Omron Sysmac Studio project Trabalho_Pratico1_vFinal_beta (Sysmac Studio 1.53.0.64009, StandardProject)

# Controller new_Controller_0: NX1P2-9B24DT1 version 1.42
Task PrimaryTask (priority 4, period or condition 4000): Tp1Automacao
Library OEN_Communication_V1_0_22 1.0.22 (contents left out)

VAR_GLOBAL RETAIN
    OutputsDigitais AT %D0 : ARRAY[0..150] OF BOOL;  (* Saidas Digitais; published *)
    DigitaInputs AT %D30 : ARRAY[0..150] OF BOOL;  (* Entradas Digitais; published *)
    AnalogInputs AT %D60 : ARRAY[0..25] OF WORD;  (* Entradas Analogicas; published *)
    AnalogOutput AT %D200 : ARRAY[0..25] OF WORD;  (* Saidas Analogicas; published *)
    Trama AT %D400 : ARRAY[0..5] OF OEN\Modbus\sModbusReq := [(Enable := True, NodeAdr := 1, FunctionCode := Fn02_ReadDiscreteInputs, Read := (StartAddressRemote := 0, StartAddressLocal := 0, Count := 35), Write := (StartAddressRemote := 0, StartAddressLocal := 0, Count := 0)), (Enable := False, NodeAdr := 1, FunctionCode := Fn05_WriteSingleCoil, Read := (StartAddressRemote := 0, StartAddressLocal := 0, Count := 0), Write := (StartAddressRemote := 0, StartAddressLocal := 0, Count := 40)), (Enable := True, NodeAdr := 1, FunctionCode := Fn15_WriteMultipleCoils, Read := (StartAddressRemote := 0, StartAddressLocal := 0, Count := 0), Write := (StartAddressRemote := 0, StartAddressLocal := 0, Count := 40)), (Enable := False, NodeAdr := 1, FunctionCode := Fn03_ReadHoldingRegisters, Read := (StartAddressRemote := 0, StartAddressLocal := 0, Count := 20), Write := (StartAddressRemote := 0, StartAddressLocal := 0, Count := 0)), (Enable := True, NodeAdr := 1, FunctionCode := Fn16_WriteMultipleRegisters, Read := (StartAddressRemote := 0, StartAddressLocal := 0, Count := 0), Write := (StartAddressRemote := 0, StartAddressLocal := 0, Count := 11)), (Enable := True, NodeAdr := 1, FunctionCode := Fn04_ReadInputRegisters, Read := (StartAddressRemote := 0, StartAddressLocal := 0, Count := 5), Write := (StartAddressRemote := 0, StartAddressLocal := 0, Count := 0))];  (* Trama de Comunicacao; published *)
END_VAR
VAR_GLOBAL
    Emerg_But : BOOL;  (* Botao de Emergencia; at BuiltInIO://cpu/#0/Input_Bit_01 *)
    Led_Is_On : BOOL;  (* Led Verde de Producao em Curso; at BuiltInIO://cpu/#0/Output_Bit_00 *)
    Start_But : BOOL;  (* Botao de início de linha; at BuiltInIO://cpu/#0/Input_Bit_02 *)
    Led_Is_Stop : BOOL;  (* Led Vermelho de linha parada; at BuiltInIO://cpu/#0/Output_Bit_01 *)
    Stop_But : BOOL;  (* Botao Stop- pára linha depois da caixa/peça ser removida; at BuiltInIO://cpu/#0/Input_Bit_03 *)
    Led_Is_Emergency : BOOL;  (* Led Amarelo de Emergência Ativa; at BuiltInIO://cpu/#0/Output_Bit_02 *)
    But_papel : BOOL;  (* Emite caixas de papel; at BuiltInIO://cpu/#0/Input_Bit_04 *)
    But_pecas : BOOL;  (* Emite peças azuis; at BuiltInIO://cpu/#0/Input_Bit_05 *)
    Sensor_IR : BOOL;  (* Sensor Infra Vermelho; at BuiltInIO://cpu/#0/Input_Bit_00 *)
    But_Reset : BOOL;  (* Reset aos contadores; at BuiltInIO://cpu/#0/Input_Bit_06 *)
    hmi_led_is_on AT %W0.00 : BOOL;  (* Led verde produção em curso; published *)
    hmi_led_is_emerg AT %W0.01 : BOOL;  (* Led amarelo de emergência; published *)
    hmi_led_is_stop AT %W0.02 : BOOL;  (* Led vermelho de linha parada; published *)
    hmi_StartBut AT %W0.03 : BOOL;  (* Botão Start- inicia linha; published *)
    hmi_StopBut AT %W0.04 : BOOL;  (* Botão Stop - pára linha depois da caixa/peça ser removida; published *)
    hmi_EmergBut AT %W0.05 : BOOL;  (* Botão Emergência - pára linha de imediato; published *)
    hmi_led_caixas AT %W0.06 : BOOL;  (* Led indica emissão de caixas de papel; published *)
    hmi_led_peças AT %W0.07 : BOOL;  (* Led indica emisão de peças azuis; published *)
    hmi_sw_emissor AT %W0.08 : BOOL;  (* Switch que emite peças (SW=0) ou caixas (SW=1); published *)
    hmi_resetCounter AT %W0.09 : BOOL;  (* Botão que dá reset aos contadores; published *)
    hmi_sw_kuka AT %W0.10 : BOOL;  (* SW=0 KUKA transforma peças em Base/ SW=1 "..."peças Lid; published *)
END_VAR
VAR_GLOBAL RETAIN
    hmi_pesoCaixa AT %D710 : INT;  (* Mostra peso da caixa; published *)
    hmi_alturaCaixa AT %D711 : INT;  (* Mostra altura da caixa; published *)
    hmi_Counter_Lid AT %D712 : INT;  (* Mosrador de peças Lid; published *)
    hmi_Counter_Base AT %D713 : INT;  (* Mostrador de peças Base; published *)
    hmi_Counter_S AT %D714 : INT;  (* Mostrador caixas S; published *)
    hmi_Counter_M AT %D715 : INT;  (* Mostrador caixas M; published *)
    hmi_Counter_L AT %D716 : INT;  (* Mostrador caixas L; published *)
END_VAR

PROGRAM Tp1Automacao
VAR
    Contact_Auxiliar : BOOL;  (* Active ad Desactive MODBUS *)
    Communication_Factory_IO : OEN\Modbus\ModbusTCP_Client;
    Etapas : INT := 0;  (* Etapas do Projeto *)
    timer_S4 : TON;  (* Permite uma leitura estável do valor medido na balança *)
END_VAR
VAR CONSTANT
    pesoCaixa_Ref : INT := 4;  (* Referencia de peso *)
END_VAR
VAR
    timer_S5 : TON;
END_VAR
VAR CONSTANT
    RightPP_Caixa1 : WORD := 8;  (* Posição em Volt para descer a Pick and Place *)
END_VAR
VAR
    timer_S6 : TON;
END_VAR
VAR RETAIN
    pesoCaixa : WORD;  (* guarda o valor do peso registado na balança *)
    pesoGuarda AT %D700 : INT;  (* Valor lido na balança em int *)
END_VAR
VAR
    ZaxisSetpoint_RightPP : WORD := 0;  (* Valor de referencia para descer o eixo Z da PP da Direita *)
    ZaxisSetpoint_KukaPP : WORD := 0;  (* Valor de referencia para descer o eixo Z da PP da kuka *)
END_VAR
VAR RETAIN
    alturaCaixa : WORD;  (* leitura o valor do altura *)
    alturaGuarda AT %D702 : INT;  (* guarda o valor da altura *)
END_VAR
VAR CONSTANT
    alturaCaixaRefM : INT := 192;  (* valor de ref para a caixa tamanho M *)
    alturaCaixaRefS : INT := 128;  (* valor de referencia para uma caixa de tamanho S (palletizing box) *)
    alturaCaixaRefL : INT := 224;  (* valor de referencia para uma caixa de tamanho L *)
    pesoCaixa_RefSmall : INT := 224;  (* ELIMINAR ESTA VARIAVEL *)
END_VAR
VAR
    timer_S7 : TON;  (* Tempo de Etiquetagem da Pick&Place Direita *)
    esteiraVel : WORD;  (* velocidade da esteira *)
    sensorVisaoLer : WORD;  (* Leitura do sensor de visão *)
END_VAR
VAR RETAIN
    sensorVisaoGuarda AT %D703 : INT;  (* guarda o valor do sensor de visao *)
END_VAR
VAR CONSTANT
    sensorVisaoRefLid : INT := 2;  (* Valor de referencia para uma tampa *)
    sensorVisaoRefRaw : INT := 1;  (* Valor de referencia para raw material *)
    sensorVisaoRefBase : INT := 3;  (* Valor de referencia para base *)
END_VAR
VAR RETAIN
    SBoxCountAux AT %D704 : INT := 0;  (* Contador de Caixas S *)
END_VAR
VAR
    SBoxCount : WORD;  (* Contador de Caixas S Para Automato *)
END_VAR
VAR RETAIN
    MBoxCountAux AT %D705 : INT := 0;  (* Contador de caixas M *)
END_VAR
VAR
    MBoxCount : WORD;  (* Contador de Caixas M Para Automato *)
END_VAR
VAR RETAIN
    LBoxCountAux AT %D706 : INT := 0;  (* Contador de caixas L *)
END_VAR
VAR
    LBoxCount : WORD;  (* Contador de Caixas L Para Automato *)
    timer_S8 : TON;  (* Tempo de atividade do Remover de Caixas S *)
    timer_S9 : TON;  (* Tempo de atividade do Remover de Caixas M *)
    timer_S10 : TON;  (* Tempo de atividade do Remover de Caixas L *)
END_VAR
VAR RETAIN
    ultimaEtapa AT %D707 : INT;  (* Variavel para guardar a ultima etapa *)
END_VAR
VAR
    ZaxisSetpoint_LeftPP : WORD := 0;  (* Valor de referencia para descer o eixo Z da PP da esquerda *)
    XaxisSetpoint_KukaPP : WORD := 0;  (* Movimento em X da pick and place *)
    timer_S11 : TON;  (* Tempo de Etiquetagem da Pick&Place Esquerda *)
END_VAR
VAR RETAIN
    LidCountAux AT %D708 : INT := 0;  (* Contador de Tampas *)
END_VAR
VAR
    LidCount : WORD;  (* Contador de Tampas para o LCD *)
END_VAR
VAR RETAIN
    BaseCountAux AT %D709 : INT := 0;  (* Contador de peças da base *)
END_VAR
VAR
    BaseCount : WORD;  (* Contador de peças base para o LCD *)
    timer_S12 : TON;  (* Tempo de atividade do Remover de Peças Lid *)
    timer_S13 : TON;  (* Tempo de atividade do Remover de Peças Base *)
    kukaSelect : INT := 0;
    ZaxisPosition_KukaPP : WORD := 0;
    XaxisPosition_KukaPP : WORD := 0;  (* Posição atual da Pick and Place da KUKA no eixo do X *)
    guardaPosZKuka : INT := 0;  (* Guarda o valor da PP da Kuka no eixo do Z *)
    guardaPosXKuka : INT := 0;  (* Guarda o valor da PP da Kuka no eixo do X *)
    SeletorKUKAAux : BOOL;  (* Variável que guarda o estado do seletor da KUKA *)
    timer_S14 : TON;  (* Permite a atualização de todos os contadores de materiais *)
    SeletorMaterialAux : BOOL;  (* Variável que guarda o estado do seletor de materiais (caixas= True / peças= False) *)
END_VAR
VAR_EXTERNAL
    OutputsDigitais : ARRAY[0..150] OF BOOL;  (* Saidas Digitais; [0] Emite peças azuis; [1] Conveyor de Entrada; [2] Conveyor da balança; [3] Ativador do Sorter; [5] Conveyor Direita; [4] Sorter Move para a Direita; [6] Sorter Move  para a Esquerda; [7] Conveyor da Esquerda; [8] Ativa tapete curvo direita; [9] Ativa tapete de medição de altura; [10] Pneumático caixa S; [11] Pneumático caixa M; [12] Pneumático caixa L; [13] Tapete curvo lado esquerdo; [14] Tapete zona de visão; [15] Vira o sorter para o raw material; [17] Vira o sorter para lid; [19] Vira o sorter para base; [16] Ativa o sorter para raw material; [18] Ativa o sorter para lid; [20] Ativa o sorter para base; [21] Tapete para a zona de separação peças; [24] Remover Caixas L; [23] Remover as Caixas do tamanho M; [22] Remover as caixas de tamanho S; [25] Conveyor de Transporte para KUKA; [27] Remover peças do tipo Base; [28] Remover peças do tipo Lid; [29] Emite caixas de papel; [30] Ativaçáo do Robot da KUKA; [31] Paragem do Robot da KUKA; [32] Conveyor Curvo da saida do Robot Kuka; [35] State=1 Ativar a fabricação de Lids. State=0 Ativar a fabricação de bases.; [36] Remover bases Kuka; [34] Tapete da direita após a saída da Kuka; [38] Agarrar na peça Pick and Place Kuka; [37] Remover tampas Kuka; [33] Conveyor lado das tampas Kuka; [39] Conveyor de Saida KUKA para peças *)
    DigitaInputs : ARRAY[0..150] OF BOOL;  (* Entradas Digitais; [0] IR Entrada; [1] Entrada na balança; [11] IR para ativar o tapete do sorter; [27] Seletor para a Kuka produzir bases; [2] IR Balança Meio; [3] IR Tapete Direita; [4] Sensor no local de etiquetagem (Direita); [5] IR Tapete Esquerda; [6] Sensor no Local de Etiquetagem (Esquerda); [7] Ativa o tapete curvo do lado direito; [8] Ativa o tapete de medição de altura; [9] IR de ativação do tapete curvo lado esquerdo; [10] IR de ativação do tapete zona de visão; [15] IR do pneumático das caixas S; [16] IR do pneumático das caixas M; [17] IR do pneumático das caixas L; [18] Deteção de caixa na pick and place da direita; [12] IR_Caixa na rampa tamanho S; [14] IR_Caixa na rampa tamanho L; [13] IR_Caixa na rampa tamanho M; [19] Detecao do Item na PP da Esquerda; [20] IR de entrada do conveyor da  KUKA; [21] Sensor do contador das bases; [22] Sensor do Contador das Lids; [23] Safety Door; [24] Sensor Capacitivo para entrada de peça producao do robot KUKA; [25] Sensor Capacitivo para notificar fim de producao de peças; [26] IR ativar o tapete apos a KUKA; [28] Seletor para a Kuka produzir Lids; [29] IR de separação de peças após a Kuka; [30] Sensor de proximidade da Pick and place da KUKA; [31] IR para contar tampas na parte da KUKA; [32] IR para contar bases na parte da kuka; [34] Estado do FactoryIO (Running ou não); [33] Estado do FactoryIO (Running ou não) *)
    AnalogInputs : ARRAY[0..25] OF WORD;  (* Entradas Analogicas; [0] Ler Peso; [1] AxisZ_Pos; [2] Sensor de visão; [3] Leitura de posição atual da Pick and Place em Z; [4] Leitura de posição atual da Pick and Place em X *)
    AnalogOutput : ARRAY[0..25] OF WORD;  (* Saidas Analogicas; [0] Esteira caixas de papelão / regular velocidade; [1] Posição do eixo Z da Pick&amp;Place Direita; [2] LCD do Contador de Caixas Pequemas ; [3] LCD das Caixas de tamanho M; [4] LCD das caixas de Tamanho L; [5] Eixo Z da PP da Esquerda; [7] Remover de peças to tipo Tampa; [8] Remover de peças to tipo Base; [9] Setpoint da posição para a pick and place da kuka Z; [10] Movimento Pick and Place KUKA em X *)
    Trama : ARRAY[0..5] OF OEN\Modbus\sModbusReq;  (* Trama de Comunicacao *)
    Start_But : BOOL;  (* Botao de inicio do tapete *)
    Led_Is_On : BOOL;  (* Led Verde de indicaçao de atividade *)
    Led_Is_Stop : BOOL;  (* Linha em Paragem *)
    Stop_But : BOOL;  (* Botao de Paragem da Producao *)
    Emerg_But : BOOL;
    Led_Is_Emergency : BOOL;
    But_papel : BOOL;  (* Botão que ativa emissão de caixas de papel- NO *)
    But_pecas : BOOL;  (* Botão que ativa a emissão de peças azuis- NC *)
    Sensor_IR : BOOL;  (* Sensor fisico IR *)
    But_Reset : BOOL;
    hmi_led_is_stop : BOOL;
    hmi_led_is_on : BOOL;
    hmi_pesoCaixa : INT;
    hmi_Counter_Lid : INT;
    hmi_Counter_Base : INT;
    hmi_Counter_S : INT;
    hmi_Counter_M : INT;
    hmi_Counter_L : INT;
    hmi_sw_kuka : BOOL;
    hmi_led_caixas : BOOL;
    hmi_led_peças : BOOL;
    hmi_resetCounter : BOOL;
    hmi_StartBut : BOOL;
    hmi_StopBut : BOOL;
    hmi_sw_emissor : BOOL;
    hmi_EmergBut : BOOL;
    hmi_alturaCaixa : INT;
    hmi_led_is_emerg : BOOL;
END_VAR
VAR
    _e1 : R_TRIG;
    _p2 : BOOL;
    _p3 : BOOL;
    _p4 : BOOL;
    _p5 : BOOL;
    _e6 : R_TRIG;
    _e7 : R_TRIG;
    _e8 : R_TRIG;
    _p9 : BOOL;
    _e10 : R_TRIG;
    _e11 : R_TRIG;
    _p12 : BOOL;
    _p13 : BOOL;
END_VAR

(* Section Tp1_Comunicação: ladder, written here as Structured Text *)

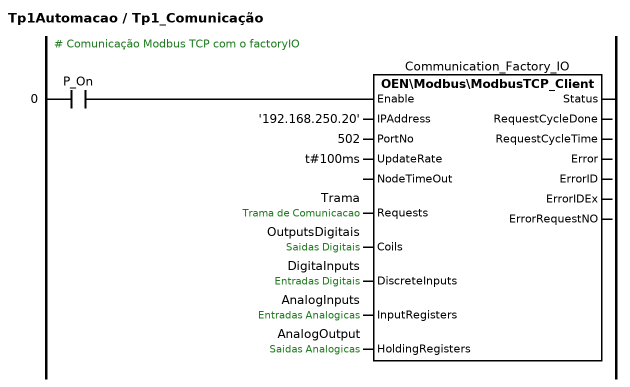
(* Rung 0: # Comunicação Modbus TCP com o factoryIO *)
Communication_Factory_IO(Enable := P_On, IPAddress := '192.168.250.20', PortNo := 502, UpdateRate := t#100ms, Requests := Trama, Coils := OutputsDigitais, DiscreteInputs := DigitaInputs, InputRegisters := AnalogInputs, HoldingRegisters := AnalogOutput);

(* Section Tp1_Botões: ladder, written here as Structured Text *)

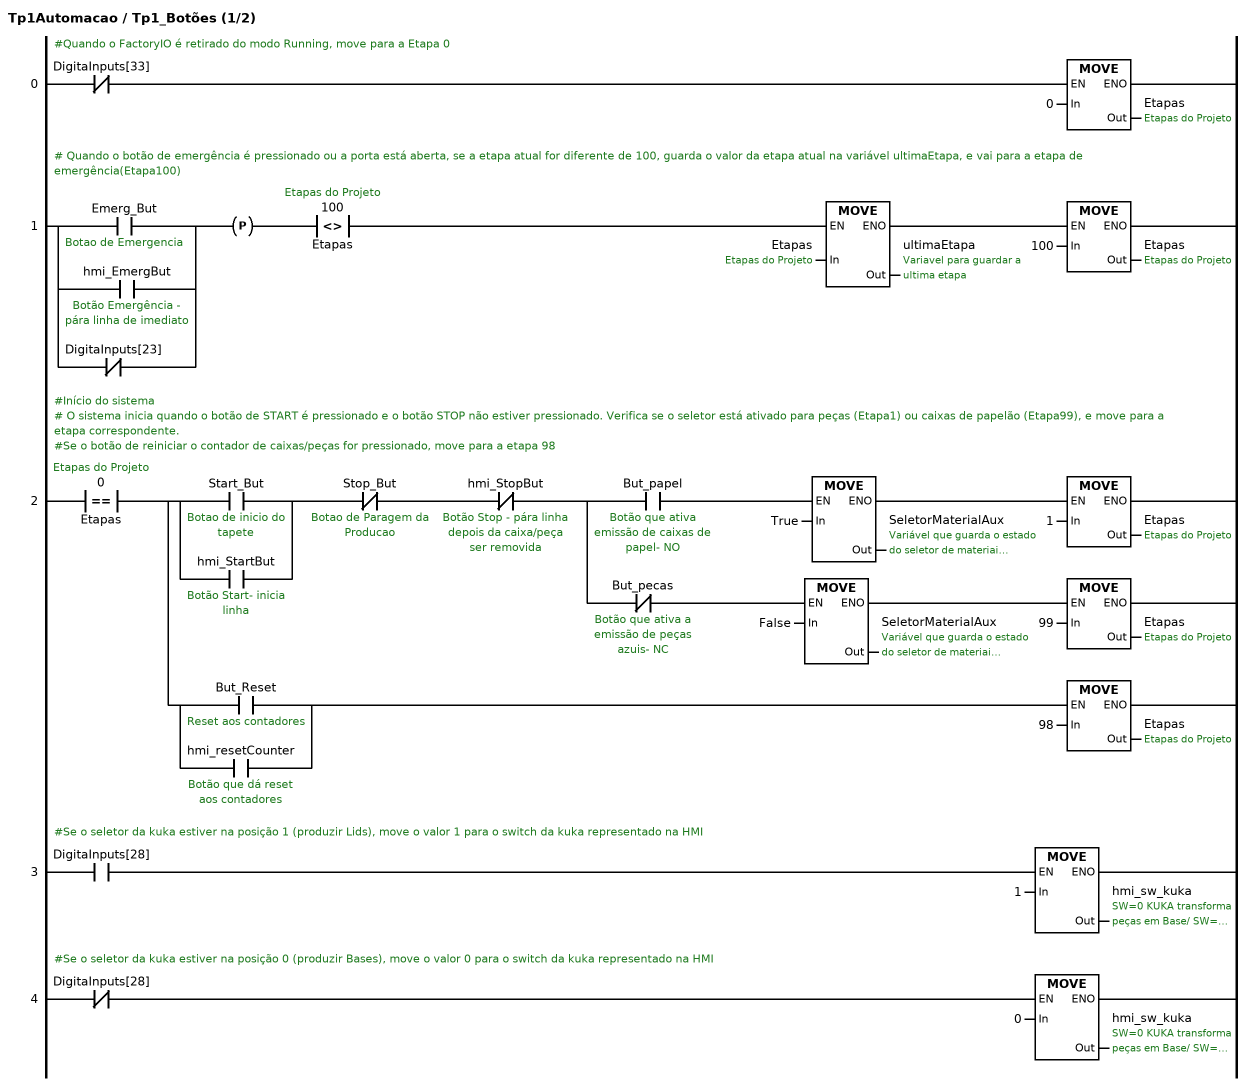
(* Rung 0: #Quando o FactoryIO é retirado do modo Running, move para a Etapa 0 *)
IF NOT DigitaInputs[33] THEN Etapas := 0; END_IF;
(* Rung 1: # Quando o botão de emergência é pressionado ou a porta está aberta, se a etapa atual for diferente de 100, guarda o valor da etapa atual na variável ultimaEtapa, e vai para a etapa de emergência(Etapa100) *)
_e1(CLK := Emerg_But OR hmi_EmergBut OR NOT DigitaInputs[23]);
IF _e1.Q AND (100 <> Etapas) THEN
    ultimaEtapa := Etapas;
    Etapas := 100;
END_IF;
(* Rung 2: #Início do sistema / # O sistema inicia quando o botão de START é pressionado e o botão STOP não estiver pressionado. Verifica se o seletor está ativado para peças (Etapa1) ou caixas de papelão (Etapa99), e move para a etapa correspondente. / #Se o botão de reiniciar o contador de caixas/peças for pressionado, move para a etapa 98 *)
_p2 := (0 = Etapas) AND (Start_But OR hmi_StartBut) AND NOT Stop_But AND NOT hmi_StopBut;
IF _p2 AND But_papel THEN SeletorMaterialAux := True; END_IF;
_p3 := 0 = Etapas;
IF _p2 AND But_papel THEN Etapas := 1; END_IF;
IF _p2 AND NOT But_pecas THEN
    SeletorMaterialAux := False;
    Etapas := 99;
END_IF;
IF _p3 AND (But_Reset OR hmi_resetCounter) THEN Etapas := 98; END_IF;
(* Rung 3: #Se o seletor da kuka estiver na posição 1 (produzir Lids), move o valor 1 para o switch da kuka representado na HMI *)
IF DigitaInputs[28] THEN hmi_sw_kuka := 1; END_IF;
(* Rung 4: #Se o seletor da kuka estiver na posição 0 (produzir Bases), move o valor 0 para o switch da kuka representado na HMI *)
IF NOT DigitaInputs[28] THEN hmi_sw_kuka := 0; END_IF;

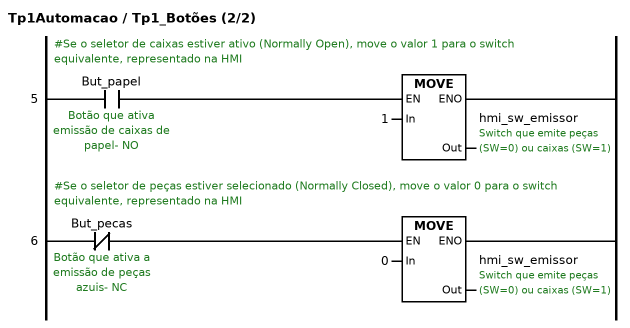
(* Rung 5: #Se o seletor de caixas estiver ativo (Normally Open), move o valor 1 para o switch equivalente, representado na HMI *)
IF But_papel THEN hmi_sw_emissor := 1; END_IF;
(* Rung 6: #Se o seletor de peças estiver selecionado (Normally Closed), move o valor 0 para o switch equivalente, representado na HMI *)
IF NOT But_pecas THEN hmi_sw_emissor := 0; END_IF;

(* Section Tp1_OutputsBotoes: ladder, written here as Structured Text *)

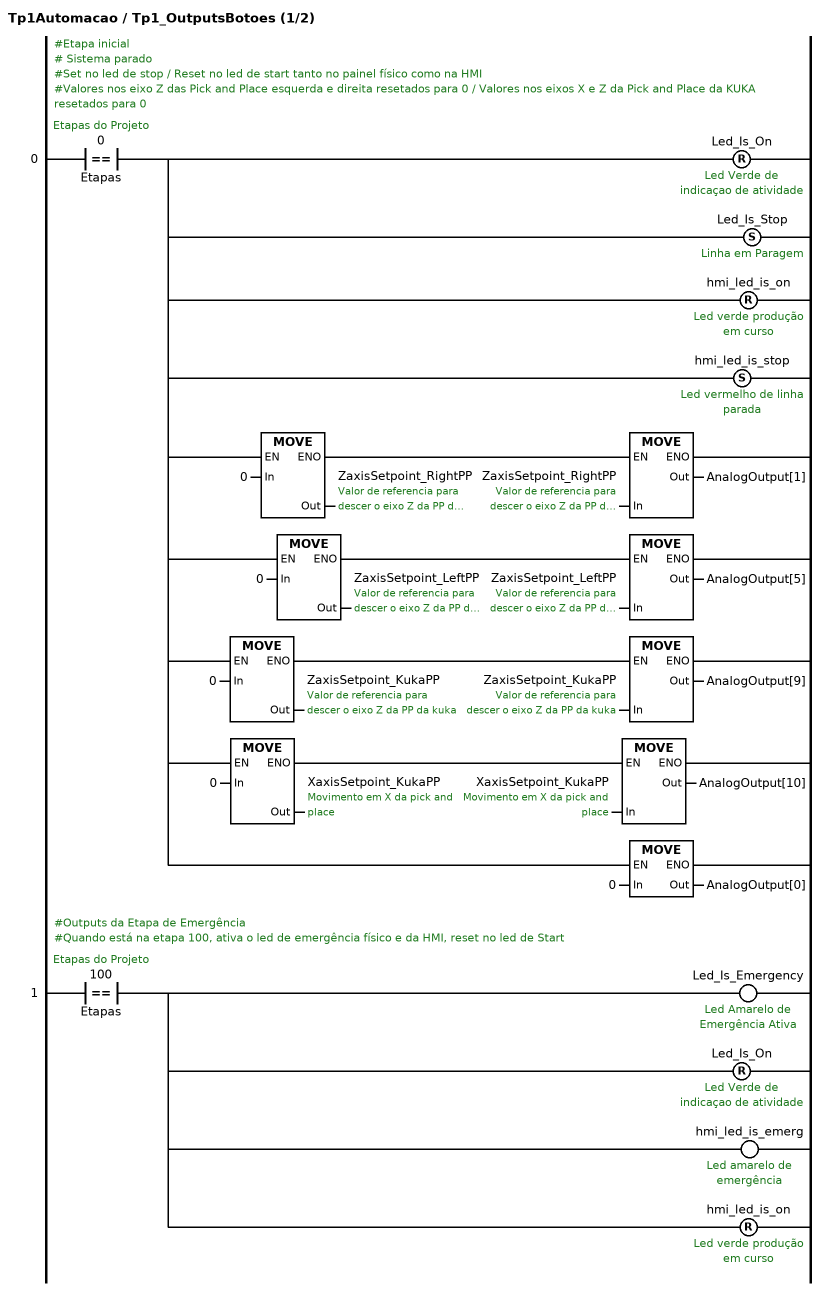
(* Rung 0: #Etapa inicial / # Sistema parado / #Set no led de stop / Reset no led de start tanto no painel físico como na HMI / #Valores nos eixo Z das Pick and Place esquerda e direita resetados para 0 / Valores nos eixos X e Z da Pick and Place da KUKA resetados para 0 *)
IF 0 = Etapas THEN
    Led_Is_On := FALSE;
    Led_Is_Stop := TRUE;
    hmi_led_is_on := FALSE;
    hmi_led_is_stop := TRUE;
    ZaxisSetpoint_RightPP := 0;
    AnalogOutput[1] := ZaxisSetpoint_RightPP;
    ZaxisSetpoint_LeftPP := 0;
    AnalogOutput[5] := ZaxisSetpoint_LeftPP;
    ZaxisSetpoint_KukaPP := 0;
    AnalogOutput[9] := ZaxisSetpoint_KukaPP;
    XaxisSetpoint_KukaPP := 0;
    AnalogOutput[10] := XaxisSetpoint_KukaPP;
    AnalogOutput[0] := 0;
END_IF;
(* Rung 1: #Outputs da Etapa de Emergência / #Quando está na etapa 100, ativa o led de emergência físico e da HMI, reset no led de Start *)
Led_Is_Emergency := 100 = Etapas;
IF 100 = Etapas THEN Led_Is_On := FALSE; END_IF;
hmi_led_is_emerg := 100 = Etapas;
IF 100 = Etapas THEN hmi_led_is_on := FALSE; END_IF;

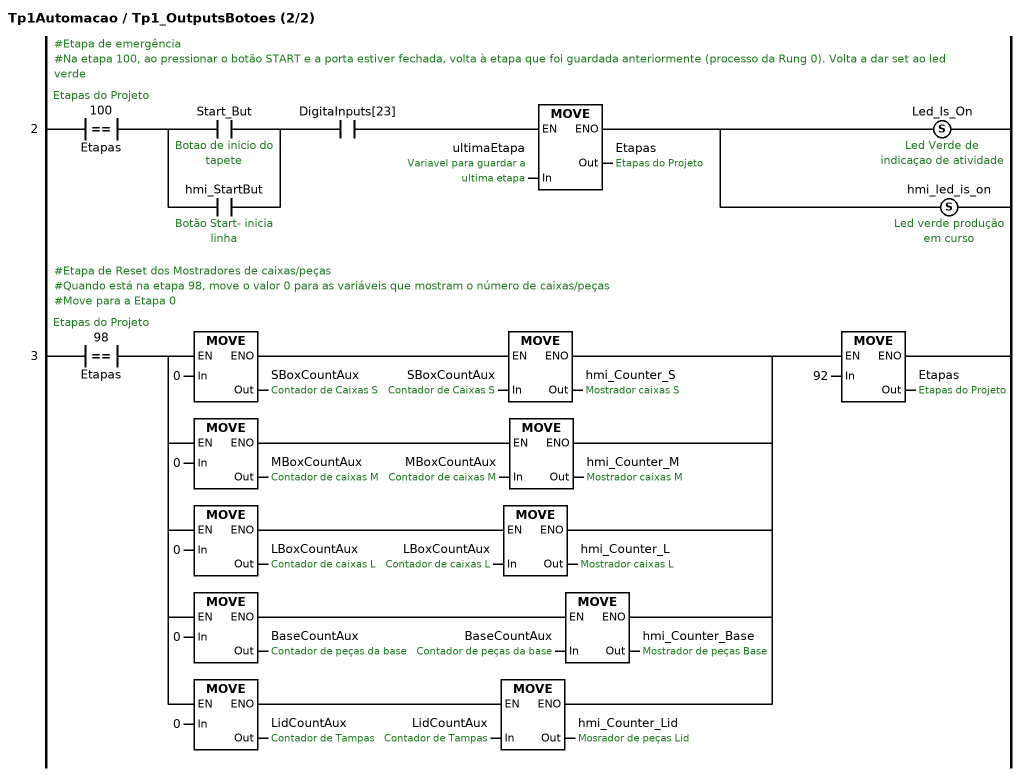
(* Rung 2: #Etapa de emergência / #Na etapa 100, ao pressionar o botão START e a porta estiver fechada, volta à etapa que foi guardada anteriormente (processo da Rung 0). Volta a dar set ao led verde *)
_p4 := (100 = Etapas) AND (Start_But OR hmi_StartBut) AND DigitaInputs[23];
IF _p4 THEN
    Etapas := ultimaEtapa;
    Led_Is_On := TRUE;
    hmi_led_is_on := TRUE;
END_IF;
(* Rung 3: #Etapa de Reset dos Mostradores de caixas/peças / #Quando está na etapa 98, move o valor 0 para as variáveis que mostram o número de caixas/peças / #Move para a Etapa 0 *)
IF 98 = Etapas THEN
    SBoxCountAux := 0;
    hmi_Counter_S := SBoxCountAux;
    MBoxCountAux := 0;
    hmi_Counter_M := MBoxCountAux;
    LBoxCountAux := 0;
    hmi_Counter_L := LBoxCountAux;
    BaseCountAux := 0;
    hmi_Counter_Base := BaseCountAux;
    LidCountAux := 0;
    hmi_Counter_Lid := LidCountAux;
    Etapas := 92;
END_IF;

(* Section Tp1_Etapas_ParteComum: ladder, written here as Structured Text *)

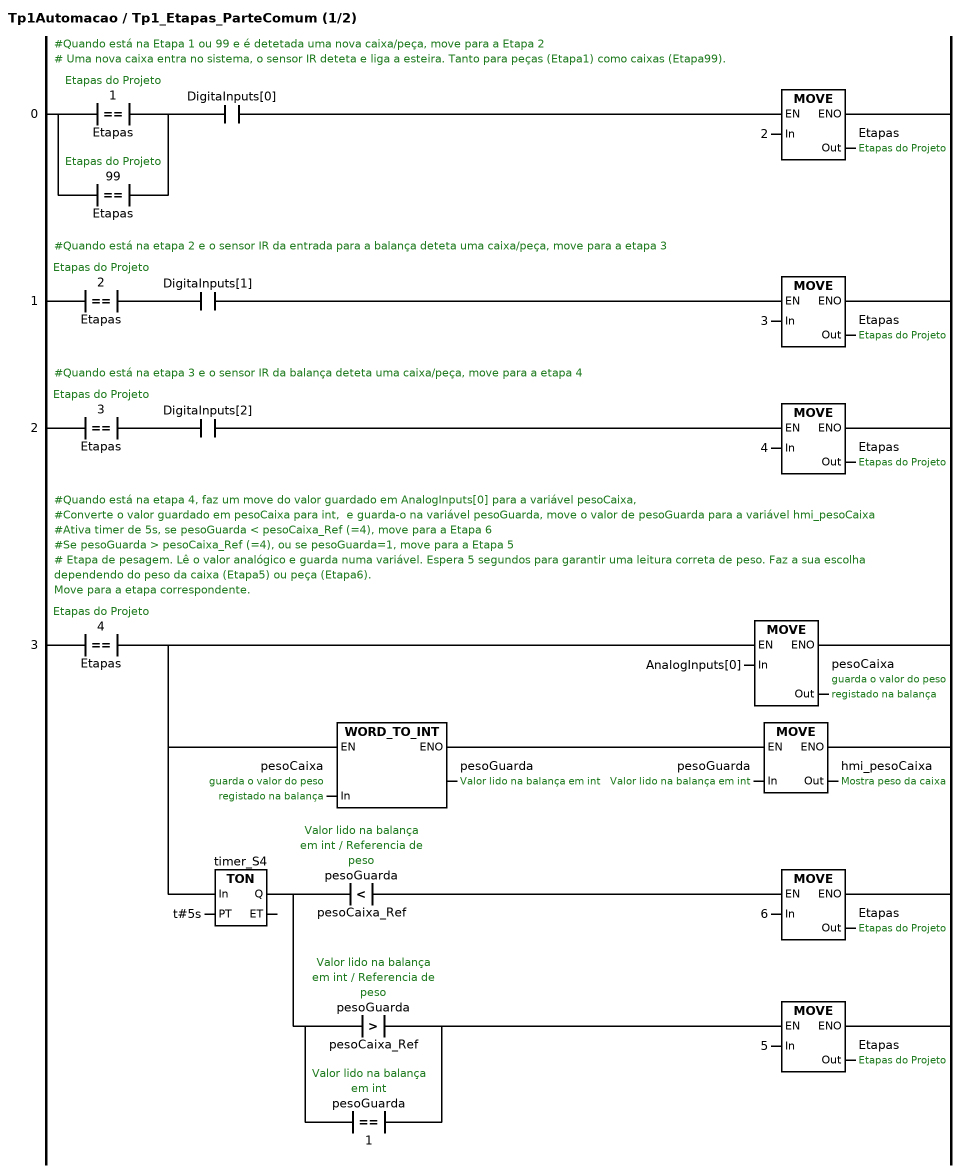
(* Rung 0: #Quando está na Etapa 1 ou 99 e é detetada uma nova caixa/peça, move para a Etapa 2 / # Uma nova caixa entra no sistema, o sensor IR deteta e liga a esteira. Tanto para peças (Etapa1) como caixas (Etapa99). *)
IF ((1 = Etapas) OR (99 = Etapas)) AND DigitaInputs[0] THEN Etapas := 2; END_IF;
(* Rung 1: #Quando está na etapa 2 e o sensor IR da entrada para a balança deteta uma caixa/peça, move para a etapa 3 *)
IF (2 = Etapas) AND DigitaInputs[1] THEN Etapas := 3; END_IF;
(* Rung 2: #Quando está na etapa 3 e o sensor IR da balança deteta uma caixa/peça, move para a etapa 4 *)
IF (3 = Etapas) AND DigitaInputs[2] THEN Etapas := 4; END_IF;
(* Rung 3: #Quando está na etapa 4, faz um move do valor guardado em AnalogInputs[0] para a variável pesoCaixa, / #Converte o valor guardado em pesoCaixa para int,  e guarda-o na variável pesoGuarda, move o valor de pesoGuarda para a variável hmi_pesoCaixa / #Ativa timer de 5s, se pesoGuarda < pesoCaixa_Ref (=4), move para a Etapa 6 / #Se pesoGuarda > pesoCaixa_Ref (=4), ou se pesoGuarda=1, move para a Etapa 5 / # Etapa de pesagem. Lê o valor analógico e guarda numa variável. Espera 5 segundos para garantir uma leitura correta de peso. Faz a sua escolha dependendo do peso da caixa (Etapa5) ou peça (Etapa6). / Move para a etapa correspondente. *)
IF 4 = Etapas THEN
    pesoCaixa := AnalogInputs[0];
    pesoGuarda := WORD_TO_INT(In := pesoCaixa);
    hmi_pesoCaixa := pesoGuarda;
END_IF;
timer_S4(In := 4 = Etapas, PT := t#5s);
IF timer_S4.Q AND (pesoGuarda < pesoCaixa_Ref) THEN Etapas := 6; END_IF;
IF timer_S4.Q AND ((pesoGuarda > pesoCaixa_Ref) OR (pesoGuarda = 1)) THEN Etapas := 5; END_IF;
(* notes on elements: #Permite a atualização de todos os contadores de materiais *)

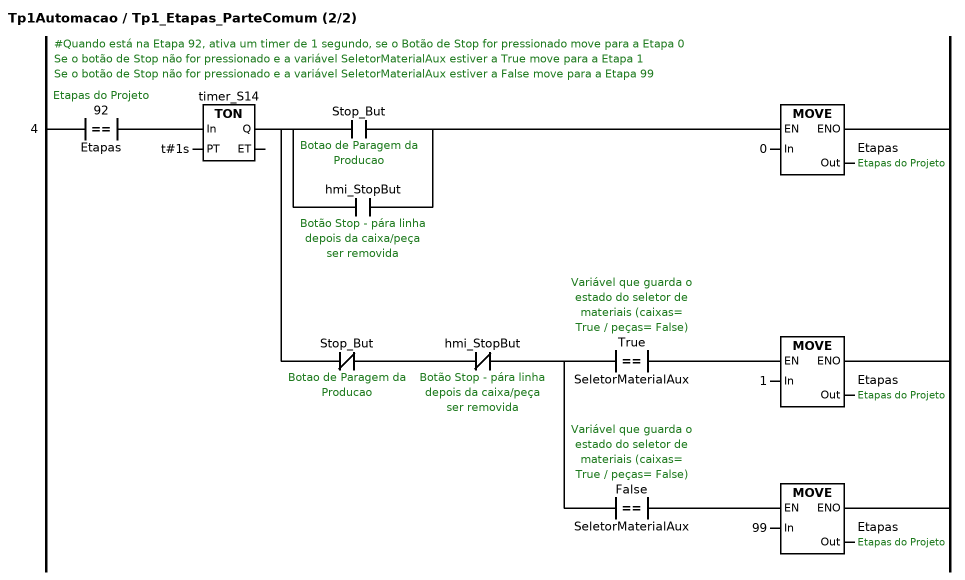
(* Rung 4: #Quando está na Etapa 92, ativa um timer de 1 segundo, se o Botão de Stop for pressionado move para a Etapa 0 / Se o botão de Stop não for pressionado e a variável SeletorMaterialAux estiver a True move para a Etapa 1 / Se o botão de Stop não for pressionado e a variável SeletorMaterialAux estiver a False move para a Etapa 99 *)
timer_S14(In := 92 = Etapas, PT := t#1s);
IF timer_S14.Q AND (Stop_But OR hmi_StopBut) THEN Etapas := 0; END_IF;
IF timer_S14.Q AND NOT Stop_But AND NOT hmi_StopBut AND (True = SeletorMaterialAux) THEN
    Etapas := 1;
END_IF;
IF timer_S14.Q AND NOT Stop_But AND NOT hmi_StopBut AND (False = SeletorMaterialAux) THEN
    Etapas := 99;
END_IF;
(* notes on elements: #Permite uma leitura estável do valor medido na balança *)

(* Section Tp1_Outputs_ParteComum: ladder, written here as Structured Text *)

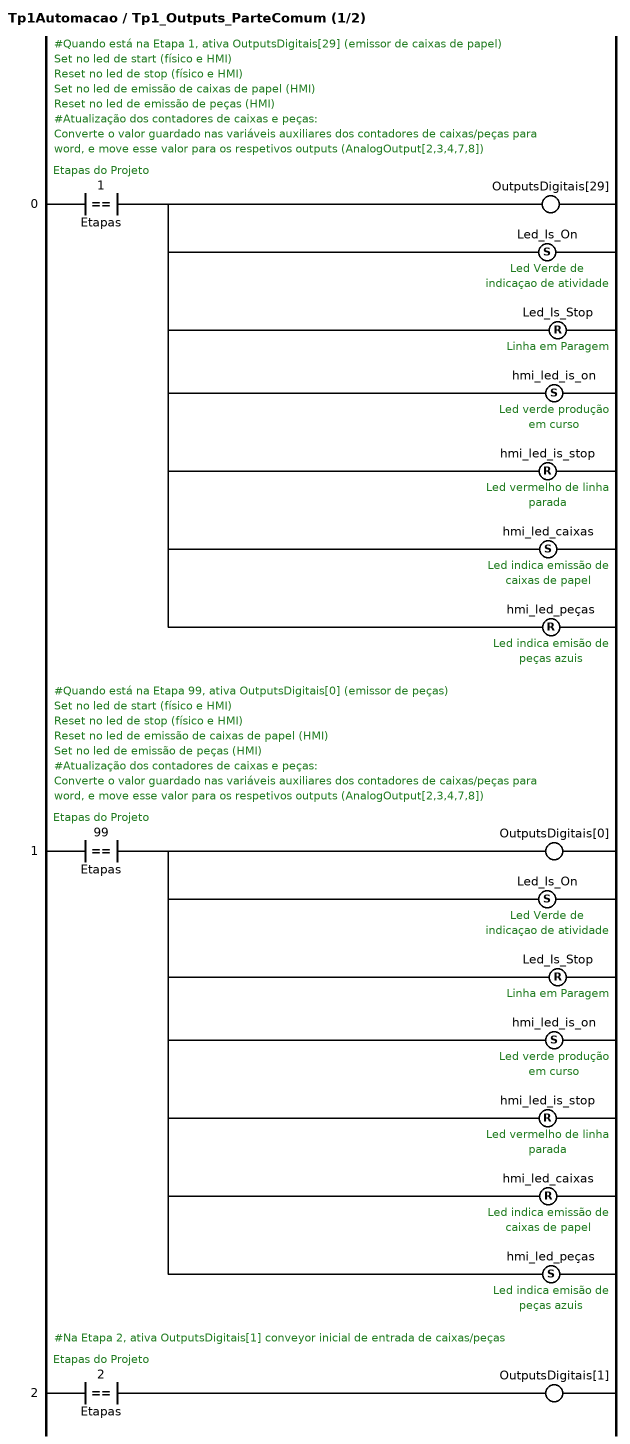
(* Rung 0: #Quando está na Etapa 1, ativa OutputsDigitais[29] (emissor de caixas de papel) / Set no led de start (físico e HMI) / Reset no led de stop (físico e HMI) / Set no led de emissão de caixas de papel (HMI) / Reset no led de emissão de peças (HMI) / #Atualização dos contadores de caixas e peças: / Converte o valor guardado nas variáveis auxiliares dos contadores de caixas/peças para word, e move esse valor para os respetivos outputs (AnalogOutput[2,3,4,7,8]) *)
OutputsDigitais[29] := 1 = Etapas;
IF 1 = Etapas THEN
    Led_Is_On := TRUE;
    Led_Is_Stop := FALSE;
    hmi_led_is_on := TRUE;
    hmi_led_is_stop := FALSE;
    hmi_led_caixas := TRUE;
    hmi_led_peças := FALSE;
END_IF;
(* Rung 1: #Quando está na Etapa 99, ativa OutputsDigitais[0] (emissor de peças) / Set no led de start (físico e HMI) / Reset no led de stop (físico e HMI) / Reset no led de emissão de caixas de papel (HMI) / Set no led de emissão de peças (HMI) / #Atualização dos contadores de caixas e peças: / Converte o valor guardado nas variáveis auxiliares dos contadores de caixas/peças para word, e move esse valor para os respetivos outputs (AnalogOutput[2,3,4,7,8]) *)
OutputsDigitais[0] := 99 = Etapas;
IF 99 = Etapas THEN
    Led_Is_On := TRUE;
    Led_Is_Stop := FALSE;
    hmi_led_is_on := TRUE;
    hmi_led_is_stop := FALSE;
    hmi_led_caixas := FALSE;
    hmi_led_peças := TRUE;
END_IF;
(* Rung 2: #Na Etapa 2, ativa OutputsDigitais[1] conveyor inicial de entrada de caixas/peças *)
OutputsDigitais[1] := 2 = Etapas;

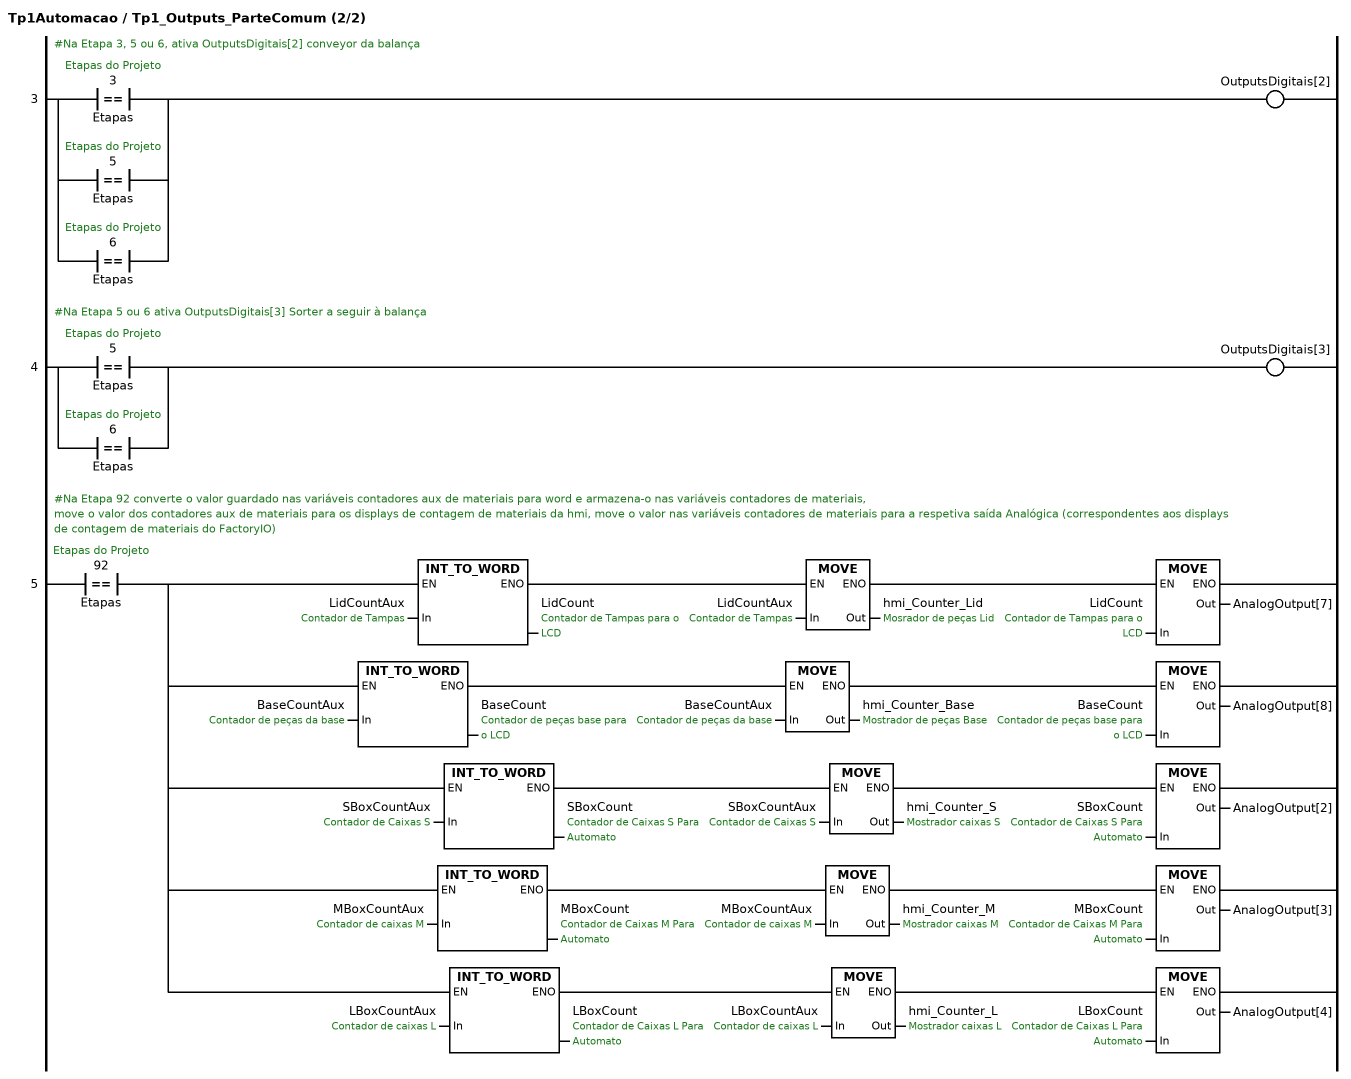
(* Rung 3: #Na Etapa 3, 5 ou 6, ativa OutputsDigitais[2] conveyor da balança *)
OutputsDigitais[2] := (3 = Etapas) OR (5 = Etapas) OR (6 = Etapas);
(* Rung 4: #Na Etapa 5 ou 6 ativa OutputsDigitais[3] Sorter a seguir à balança *)
OutputsDigitais[3] := (5 = Etapas) OR (6 = Etapas);
(* Rung 5: #Na Etapa 92 converte o valor guardado nas variáveis contadores aux de materiais para word e armazena-o nas variáveis contadores de materiais, / move o valor dos contadores aux de materiais para os displays de contagem de materiais da hmi, move o valor nas variáveis contadores de materiais para a respetiva saída Analógica (correspondentes aos displays / de contagem de materiais do FactoryIO) *)
IF 92 = Etapas THEN
    LidCount := INT_TO_WORD(In := LidCountAux);
    hmi_Counter_Lid := LidCountAux;
    AnalogOutput[7] := LidCount;
    BaseCount := INT_TO_WORD(In := BaseCountAux);
    hmi_Counter_Base := BaseCountAux;
    AnalogOutput[8] := BaseCount;
    SBoxCount := INT_TO_WORD(In := SBoxCountAux);
    hmi_Counter_S := SBoxCountAux;
    AnalogOutput[2] := SBoxCount;
    MBoxCount := INT_TO_WORD(In := MBoxCountAux);
    hmi_Counter_M := MBoxCountAux;
    AnalogOutput[3] := MBoxCount;
    LBoxCount := INT_TO_WORD(In := LBoxCountAux);
    hmi_Counter_L := LBoxCountAux;
    AnalogOutput[4] := LBoxCount;
END_IF;

(* Section Tp1_Etapas_ParteDireita: ladder, written here as Structured Text *)

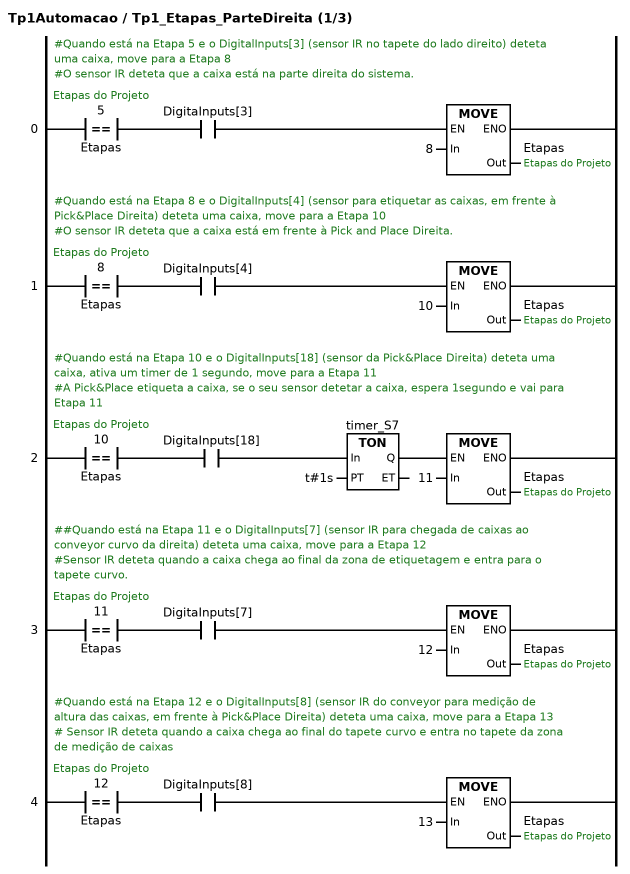
(* Rung 0: #Quando está na Etapa 5 e o DigitalInputs[3] (sensor IR no tapete do lado direito) deteta uma caixa, move para a Etapa 8 / #O sensor IR deteta que a caixa está na parte direita do sistema. *)
IF (5 = Etapas) AND DigitaInputs[3] THEN Etapas := 8; END_IF;
(* Rung 1: #Quando está na Etapa 8 e o DigitalInputs[4] (sensor para etiquetar as caixas, em frente à Pick&Place Direita) deteta uma caixa, move para a Etapa 10 / #O sensor IR deteta que a caixa está em frente à Pick and Place Direita. *)
IF (8 = Etapas) AND DigitaInputs[4] THEN Etapas := 10; END_IF;
(* Rung 2: #Quando está na Etapa 10 e o DigitalInputs[18] (sensor da Pick&Place Direita) deteta uma caixa, ativa um timer de 1 segundo, move para a Etapa 11 / #A Pick&Place etiqueta a caixa, se o seu sensor detetar a caixa, espera 1segundo e vai para Etapa 11 *)
timer_S7(In := (10 = Etapas) AND DigitaInputs[18], PT := t#1s);
IF timer_S7.Q THEN Etapas := 11; END_IF;
(* notes on elements: Tempo de Etiquetagem da Pick&Place Direita *)
(* Rung 3: ##Quando está na Etapa 11 e o DigitalInputs[7] (sensor IR para chegada de caixas ao conveyor curvo da direita) deteta uma caixa, move para a Etapa 12 / #Sensor IR deteta quando a caixa chega ao final da zona de etiquetagem e entra para o tapete curvo. *)
IF (11 = Etapas) AND DigitaInputs[7] THEN Etapas := 12; END_IF;
(* Rung 4: #Quando está na Etapa 12 e o DigitalInputs[8] (sensor IR do conveyor para medição de altura das caixas, em frente à Pick&Place Direita) deteta uma caixa, move para a Etapa 13 / # Sensor IR deteta quando a caixa chega ao final do tapete curvo e entra no tapete da zona de medição de caixas *)
IF (12 = Etapas) AND DigitaInputs[8] THEN Etapas := 13; END_IF;

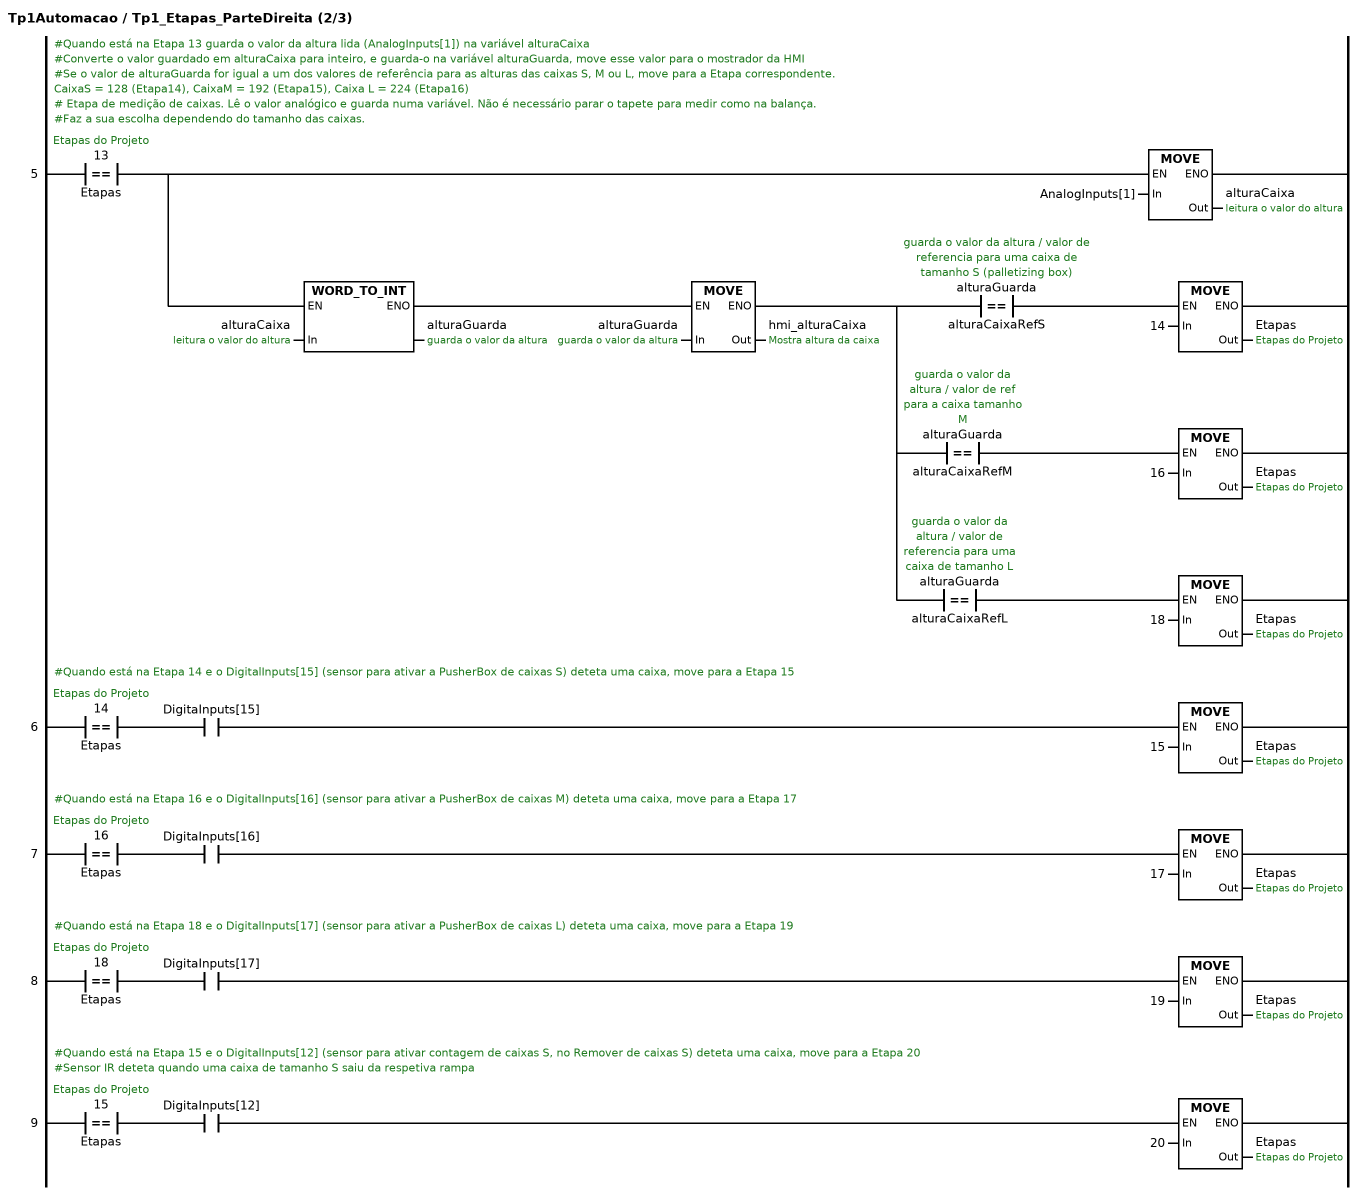
(* Rung 5: #Quando está na Etapa 13 guarda o valor da altura lida (AnalogInputs[1]) na variável alturaCaixa / #Converte o valor guardado em alturaCaixa para inteiro, e guarda-o na variável alturaGuarda, move esse valor para o mostrador da HMI / #Se o valor de alturaGuarda for igual a um dos valores de referência para as alturas das caixas S, M ou L, move para a Etapa correspondente. / CaixaS = 128 (Etapa14), CaixaM = 192 (Etapa15), Caixa L = 224 (Etapa16) / # Etapa de medição de caixas. Lê o valor analógico e guarda numa variável. Não é necessário parar o tapete para medir como na balança. / #Faz a sua escolha dependendo do tamanho das caixas. *)
IF 13 = Etapas THEN
    alturaCaixa := AnalogInputs[1];
    alturaGuarda := WORD_TO_INT(In := alturaCaixa);
    hmi_alturaCaixa := alturaGuarda;
END_IF;
_p5 := 13 = Etapas;
IF (13 = Etapas) AND (alturaGuarda = alturaCaixaRefS) THEN Etapas := 14; END_IF;
IF _p5 AND (alturaGuarda = alturaCaixaRefM) THEN Etapas := 16; END_IF;
IF _p5 AND (alturaGuarda = alturaCaixaRefL) THEN Etapas := 18; END_IF;
(* Rung 6: #Quando está na Etapa 14 e o DigitalInputs[15] (sensor para ativar a PusherBox de caixas S) deteta uma caixa, move para a Etapa 15 *)
IF (14 = Etapas) AND DigitaInputs[15] THEN Etapas := 15; END_IF;
(* Rung 7: #Quando está na Etapa 16 e o DigitalInputs[16] (sensor para ativar a PusherBox de caixas M) deteta uma caixa, move para a Etapa 17 *)
IF (16 = Etapas) AND DigitaInputs[16] THEN Etapas := 17; END_IF;
(* Rung 8: #Quando está na Etapa 18 e o DigitalInputs[17] (sensor para ativar a PusherBox de caixas L) deteta uma caixa, move para a Etapa 19 *)
IF (18 = Etapas) AND DigitaInputs[17] THEN Etapas := 19; END_IF;
(* Rung 9: #Quando está na Etapa 15 e o DigitalInputs[12] (sensor para ativar contagem de caixas S, no Remover de caixas S) deteta uma caixa, move para a Etapa 20 / #Sensor IR deteta quando uma caixa de tamanho S saiu da respetiva rampa *)
IF (15 = Etapas) AND DigitaInputs[12] THEN Etapas := 20; END_IF;

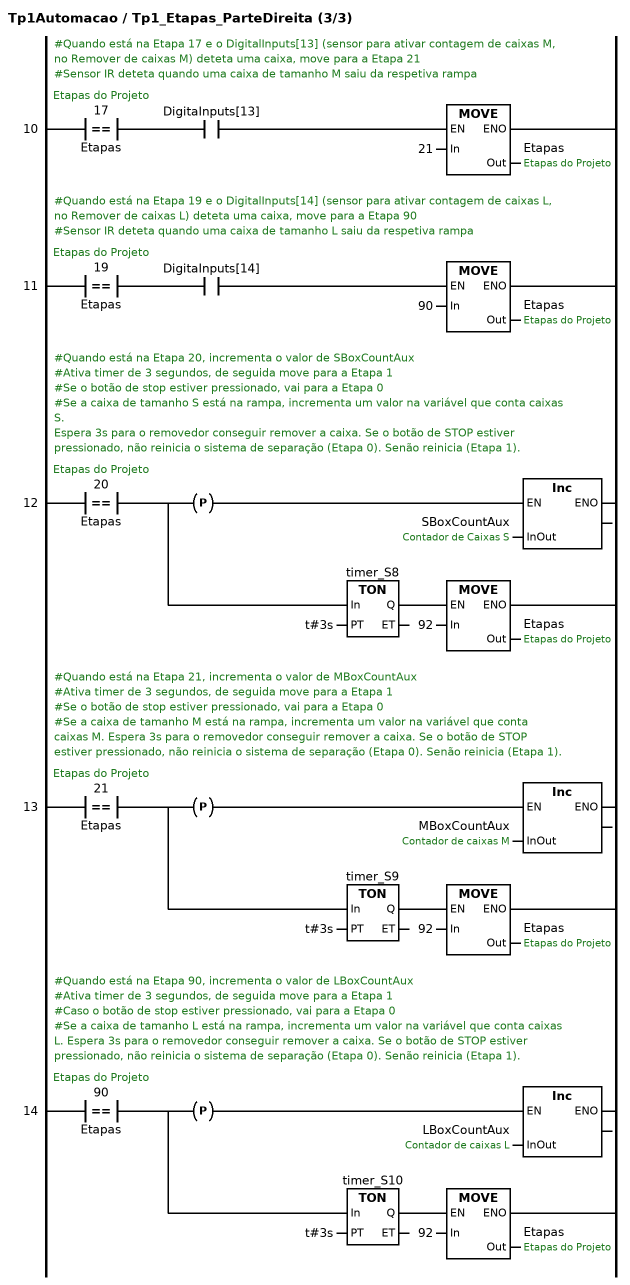
(* Rung 10: #Quando está na Etapa 17 e o DigitalInputs[13] (sensor para ativar contagem de caixas M, no Remover de caixas M) deteta uma caixa, move para a Etapa 21 / #Sensor IR deteta quando uma caixa de tamanho M saiu da respetiva rampa *)
IF (17 = Etapas) AND DigitaInputs[13] THEN Etapas := 21; END_IF;
(* Rung 11: #Quando está na Etapa 19 e o DigitalInputs[14] (sensor para ativar contagem de caixas L, no Remover de caixas L) deteta uma caixa, move para a Etapa 90 / #Sensor IR deteta quando uma caixa de tamanho L saiu da respetiva rampa *)
IF (19 = Etapas) AND DigitaInputs[14] THEN Etapas := 90; END_IF;
(* Rung 12: #Quando está na Etapa 20, incrementa o valor de SBoxCountAux / #Ativa timer de 3 segundos, de seguida move para a Etapa 1 / #Se o botão de stop estiver pressionado, vai para a Etapa 0 / #Se a caixa de tamanho S está na rampa, incrementa um valor na variável que conta caixas S. / Espera 3s para o removedor conseguir remover a caixa. Se o botão de STOP estiver pressionado, não reinicia o sistema de separação (Etapa 0). Senão reinicia (Etapa 1). *)
_e6(CLK := 20 = Etapas);
IF _e6.Q THEN Inc(InOut := SBoxCountAux); END_IF;
timer_S8(In := 20 = Etapas, PT := t#3s);
IF timer_S8.Q THEN Etapas := 92; END_IF;
(* notes on elements: Tempo de atividade do Remover de Caixas S *)
(* Rung 13: #Quando está na Etapa 21, incrementa o valor de MBoxCountAux / #Ativa timer de 3 segundos, de seguida move para a Etapa 1 / #Se o botão de stop estiver pressionado, vai para a Etapa 0 / #Se a caixa de tamanho M está na rampa, incrementa um valor na variável que conta caixas M. Espera 3s para o removedor conseguir remover a caixa. Se o botão de STOP estiver pressionado, não reinicia o sistema de separação (Etapa 0). Senão reinicia (Etapa 1). *)
_e7(CLK := 21 = Etapas);
IF _e7.Q THEN Inc(InOut := MBoxCountAux); END_IF;
timer_S9(In := 21 = Etapas, PT := t#3s);
IF timer_S9.Q THEN Etapas := 92; END_IF;
(* notes on elements: Tempo de atividade do Remover de Caixas M *)
(* Rung 14: #Quando está na Etapa 90, incrementa o valor de LBoxCountAux / #Ativa timer de 3 segundos, de seguida move para a Etapa 1 / #Caso o botão de stop estiver pressionado, vai para a Etapa 0 / #Se a caixa de tamanho L está na rampa, incrementa um valor na variável que conta caixas L. Espera 3s para o removedor conseguir remover a caixa. Se o botão de STOP estiver pressionado, não reinicia o sistema de separação (Etapa 0). Senão reinicia (Etapa 1). *)
_e8(CLK := 90 = Etapas);
IF _e8.Q THEN Inc(InOut := LBoxCountAux); END_IF;
timer_S10(In := 90 = Etapas, PT := t#3s);
IF timer_S10.Q THEN Etapas := 92; END_IF;
(* notes on elements: Tempo de atividade do Remover de Caixas L *)

(* Section Tp1_Outputs_ParteDireita: ladder, written here as Structured Text *)

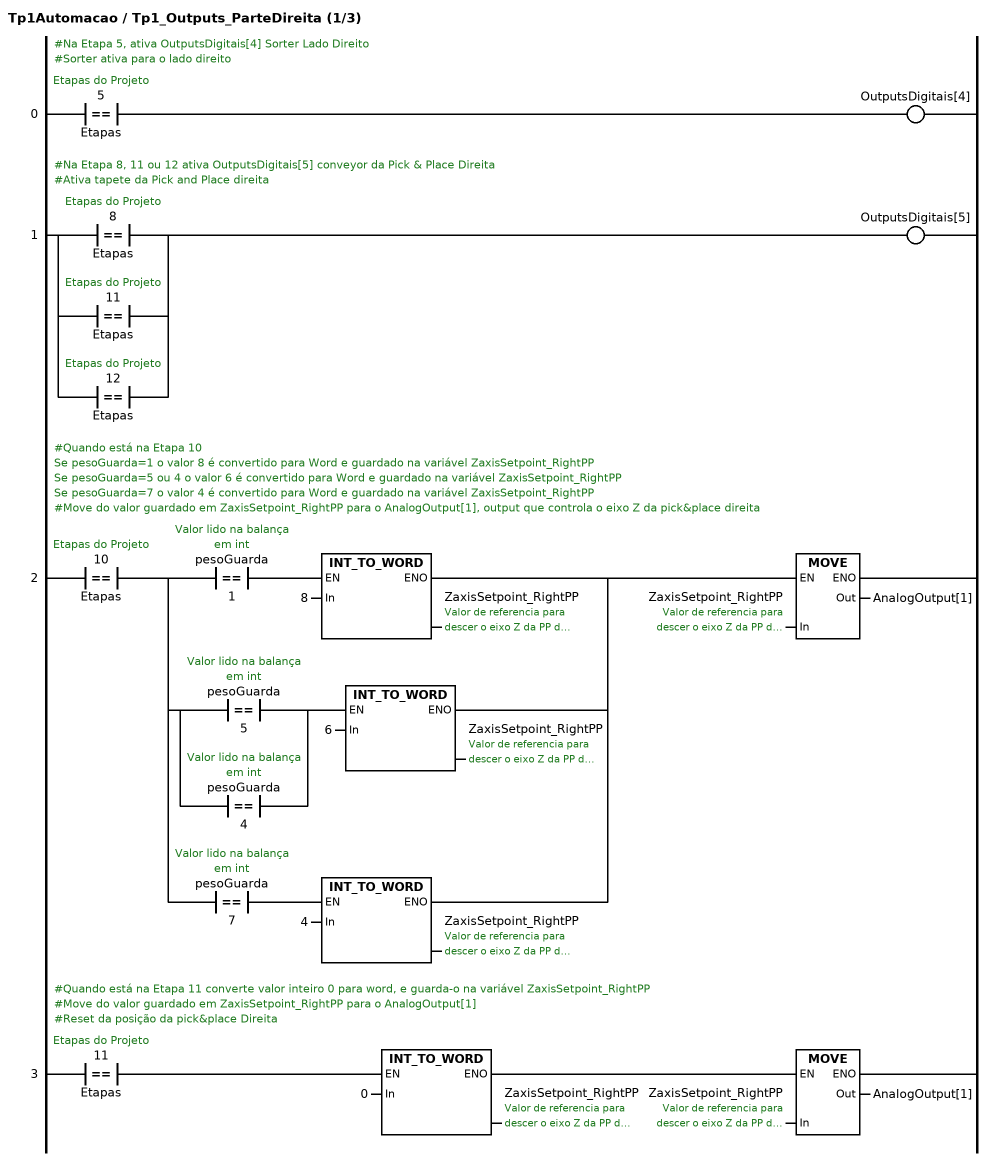
(* Rung 0: #Na Etapa 5, ativa OutputsDigitais[4] Sorter Lado Direito / #Sorter ativa para o lado direito *)
OutputsDigitais[4] := 5 = Etapas;
(* Rung 1: #Na Etapa 8, 11 ou 12 ativa OutputsDigitais[5] conveyor da Pick & Place Direita / #Ativa tapete da Pick and Place direita *)
OutputsDigitais[5] := (8 = Etapas) OR (11 = Etapas) OR (12 = Etapas);
(* Rung 2: #Quando está na Etapa 10 / Se pesoGuarda=1 o valor 8 é convertido para Word e guardado na variável ZaxisSetpoint_RightPP / Se pesoGuarda=5 ou 4 o valor 6 é convertido para Word e guardado na variável ZaxisSetpoint_RightPP / Se pesoGuarda=7 o valor 4 é convertido para Word e guardado na variável ZaxisSetpoint_RightPP / #Move do valor guardado em ZaxisSetpoint_RightPP para o AnalogOutput[1], output que controla o eixo Z da pick&place direita *)
IF (10 = Etapas) AND (pesoGuarda = 1) THEN ZaxisSetpoint_RightPP := INT_TO_WORD(In := 8); END_IF;
IF (10 = Etapas) AND ((pesoGuarda = 5) OR (pesoGuarda = 4)) THEN
    ZaxisSetpoint_RightPP := INT_TO_WORD(In := 6);
END_IF;
IF (10 = Etapas) AND (pesoGuarda = 7) THEN ZaxisSetpoint_RightPP := INT_TO_WORD(In := 4); END_IF;
IF (10 = Etapas) AND ((pesoGuarda = 1) OR (pesoGuarda = 5) OR (pesoGuarda = 4) OR (pesoGuarda = 7)) THEN
    AnalogOutput[1] := ZaxisSetpoint_RightPP;
END_IF;
(* Rung 3: #Quando está na Etapa 11 converte valor inteiro 0 para word, e guarda-o na variável ZaxisSetpoint_RightPP / #Move do valor guardado em ZaxisSetpoint_RightPP para o AnalogOutput[1] / #Reset da posição da pick&place Direita *)
IF 11 = Etapas THEN
    ZaxisSetpoint_RightPP := INT_TO_WORD(In := 0);
    AnalogOutput[1] := ZaxisSetpoint_RightPP;
END_IF;

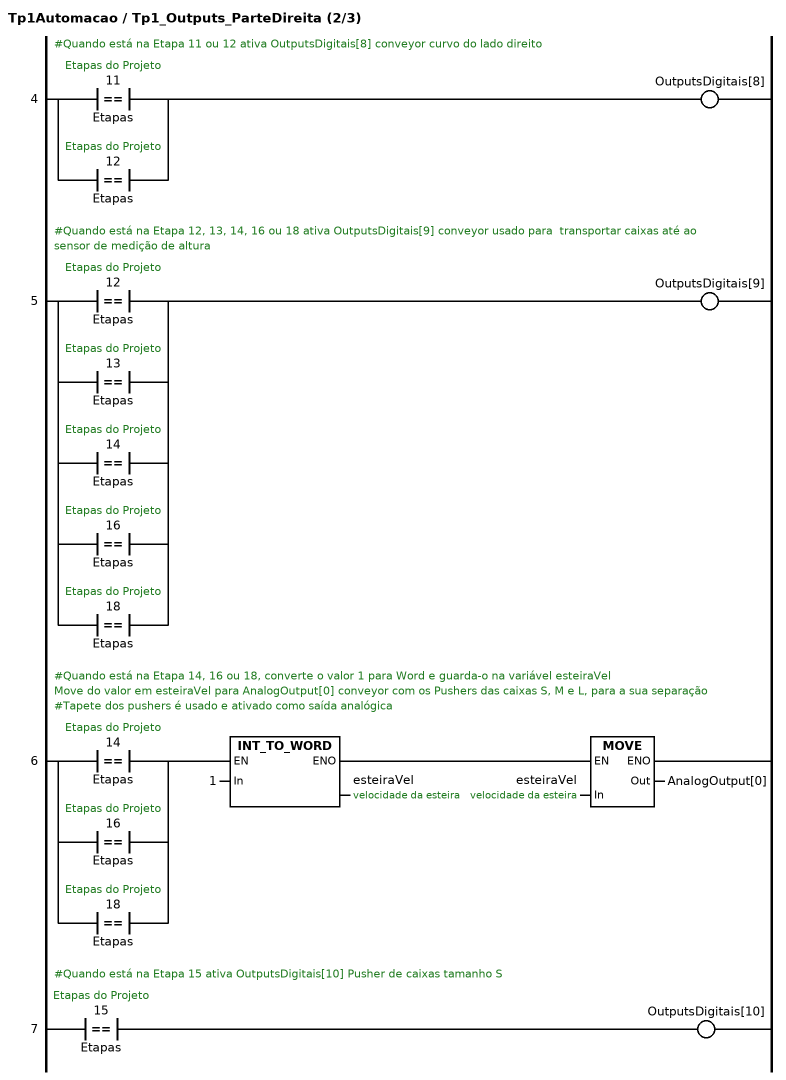
(* Rung 4: #Quando está na Etapa 11 ou 12 ativa OutputsDigitais[8] conveyor curvo do lado direito *)
OutputsDigitais[8] := (11 = Etapas) OR (12 = Etapas);
(* Rung 5: #Quando está na Etapa 12, 13, 14, 16 ou 18 ativa OutputsDigitais[9] conveyor usado para  transportar caixas até ao sensor de medição de altura *)
OutputsDigitais[9] := (12 = Etapas) OR (13 = Etapas) OR (14 = Etapas) OR (16 = Etapas) OR (18 = Etapas);
(* Rung 6: #Quando está na Etapa 14, 16 ou 18, converte o valor 1 para Word e guarda-o na variável esteiraVel / Move do valor em esteiraVel para AnalogOutput[0] conveyor com os Pushers das caixas S, M e L, para a sua separação / #Tapete dos pushers é usado e ativado como saída analógica *)
IF (14 = Etapas) OR (16 = Etapas) OR (18 = Etapas) THEN
    esteiraVel := INT_TO_WORD(In := 1);
    AnalogOutput[0] := esteiraVel;
END_IF;
(* Rung 7: #Quando está na Etapa 15 ativa OutputsDigitais[10] Pusher de caixas tamanho S *)
OutputsDigitais[10] := 15 = Etapas;

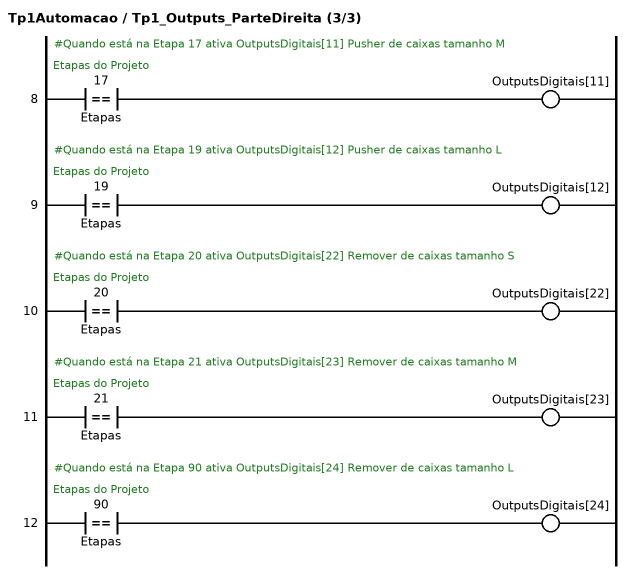
(* Rung 8: #Quando está na Etapa 17 ativa OutputsDigitais[11] Pusher de caixas tamanho M *)
OutputsDigitais[11] := 17 = Etapas;
(* Rung 9: #Quando está na Etapa 19 ativa OutputsDigitais[12] Pusher de caixas tamanho L *)
OutputsDigitais[12] := 19 = Etapas;
(* Rung 10: #Quando está na Etapa 20 ativa OutputsDigitais[22] Remover de caixas tamanho S *)
OutputsDigitais[22] := 20 = Etapas;
(* Rung 11: #Quando está na Etapa 21 ativa OutputsDigitais[23] Remover de caixas tamanho M *)
OutputsDigitais[23] := 21 = Etapas;
(* Rung 12: #Quando está na Etapa 90 ativa OutputsDigitais[24] Remover de caixas tamanho L *)
OutputsDigitais[24] := 90 = Etapas;

(* Section Tp1_Etapas_ParteEsquerda: ladder, written here as Structured Text *)

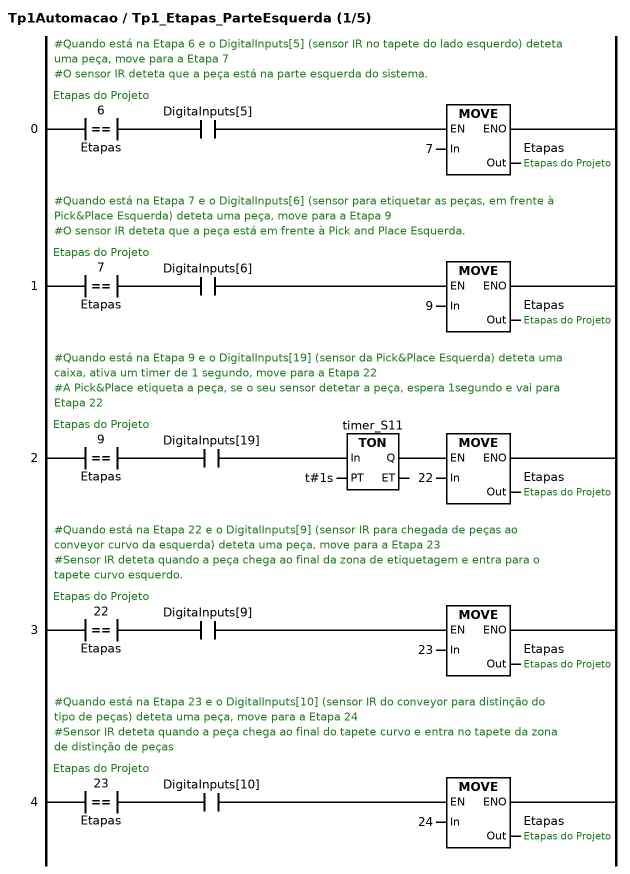
(* Rung 0: #Quando está na Etapa 6 e o DigitalInputs[5] (sensor IR no tapete do lado esquerdo) deteta uma peça, move para a Etapa 7 / #O sensor IR deteta que a peça está na parte esquerda do sistema. *)
IF (6 = Etapas) AND DigitaInputs[5] THEN Etapas := 7; END_IF;
(* Rung 1: #Quando está na Etapa 7 e o DigitalInputs[6] (sensor para etiquetar as peças, em frente à Pick&Place Esquerda) deteta uma peça, move para a Etapa 9 / #O sensor IR deteta que a peça está em frente à Pick and Place Esquerda. *)
IF (7 = Etapas) AND DigitaInputs[6] THEN Etapas := 9; END_IF;
(* Rung 2: #Quando está na Etapa 9 e o DigitalInputs[19] (sensor da Pick&Place Esquerda) deteta uma caixa, ativa um timer de 1 segundo, move para a Etapa 22 / #A Pick&Place etiqueta a peça, se o seu sensor detetar a peça, espera 1segundo e vai para Etapa 22 *)
timer_S11(In := (9 = Etapas) AND DigitaInputs[19], PT := t#1s);
IF timer_S11.Q THEN Etapas := 22; END_IF;
(* notes on elements: Tempo de Etiquetagem da Pick&Place Esquerda *)
(* Rung 3: #Quando está na Etapa 22 e o DigitalInputs[9] (sensor IR para chegada de peças ao conveyor curvo da esquerda) deteta uma peça, move para a Etapa 23 / #Sensor IR deteta quando a peça chega ao final da zona de etiquetagem e entra para o tapete curvo esquerdo. *)
IF (22 = Etapas) AND DigitaInputs[9] THEN Etapas := 23; END_IF;
(* Rung 4: #Quando está na Etapa 23 e o DigitalInputs[10] (sensor IR do conveyor para distinção do tipo de peças) deteta uma peça, move para a Etapa 24 / #Sensor IR deteta quando a peça chega ao final do tapete curvo e entra no tapete da zona de distinção de peças *)
IF (23 = Etapas) AND DigitaInputs[10] THEN Etapas := 24; END_IF;

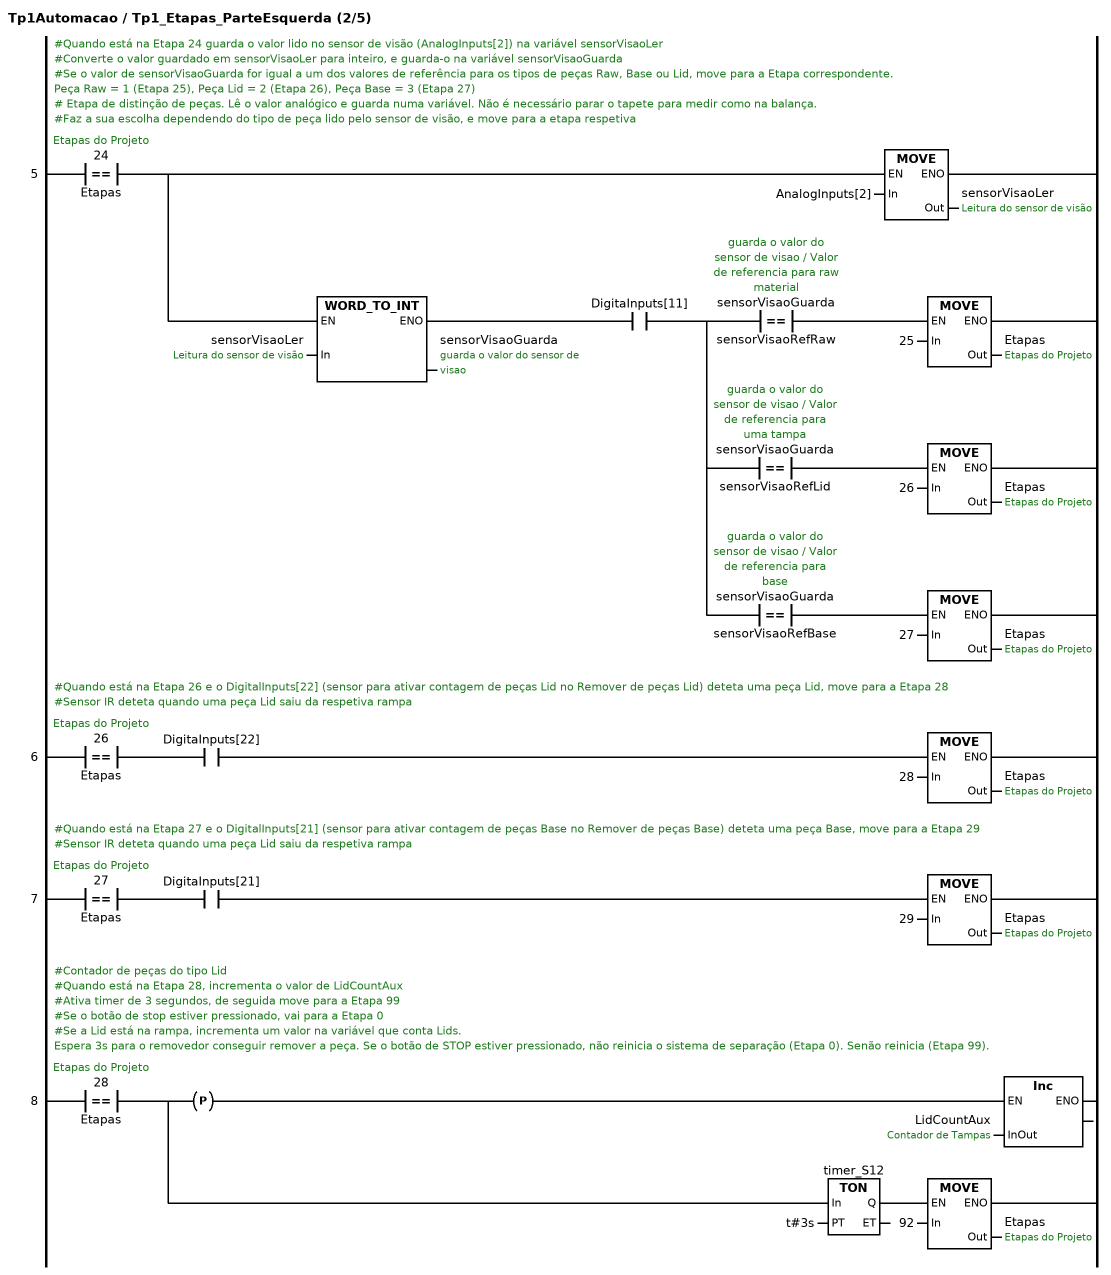
(* Rung 5: #Quando está na Etapa 24 guarda o valor lido no sensor de visão (AnalogInputs[2]) na variável sensorVisaoLer / #Converte o valor guardado em sensorVisaoLer para inteiro, e guarda-o na variável sensorVisaoGuarda / #Se o valor de sensorVisaoGuarda for igual a um dos valores de referência para os tipos de peças Raw, Base ou Lid, move para a Etapa correspondente. / Peça Raw = 1 (Etapa 25), Peça Lid = 2 (Etapa 26), Peça Base = 3 (Etapa 27) / # Etapa de distinção de peças. Lê o valor analógico e guarda numa variável. Não é necessário parar o tapete para medir como na balança. / #Faz a sua escolha dependendo do tipo de peça lido pelo sensor de visão, e move para a etapa respetiva *)
IF 24 = Etapas THEN
    sensorVisaoLer := AnalogInputs[2];
    sensorVisaoGuarda := WORD_TO_INT(In := sensorVisaoLer);
END_IF;
_p9 := (24 = Etapas) AND DigitaInputs[11];
IF (24 = Etapas) AND DigitaInputs[11] AND (sensorVisaoGuarda = sensorVisaoRefRaw) THEN
    Etapas := 25;
END_IF;
IF _p9 AND (sensorVisaoGuarda = sensorVisaoRefLid) THEN Etapas := 26; END_IF;
IF _p9 AND (sensorVisaoGuarda = sensorVisaoRefBase) THEN Etapas := 27; END_IF;
(* Rung 6: #Quando está na Etapa 26 e o DigitalInputs[22] (sensor para ativar contagem de peças Lid no Remover de peças Lid) deteta uma peça Lid, move para a Etapa 28 / #Sensor IR deteta quando uma peça Lid saiu da respetiva rampa *)
IF (26 = Etapas) AND DigitaInputs[22] THEN Etapas := 28; END_IF;
(* Rung 7: #Quando está na Etapa 27 e o DigitalInputs[21] (sensor para ativar contagem de peças Base no Remover de peças Base) deteta uma peça Base, move para a Etapa 29 / #Sensor IR deteta quando uma peça Lid saiu da respetiva rampa *)
IF (27 = Etapas) AND DigitaInputs[21] THEN Etapas := 29; END_IF;
(* Rung 8: #Contador de peças do tipo Lid / #Quando está na Etapa 28, incrementa o valor de LidCountAux / #Ativa timer de 3 segundos, de seguida move para a Etapa 99 / #Se o botão de stop estiver pressionado, vai para a Etapa 0 / #Se a Lid está na rampa, incrementa um valor na variável que conta Lids. / Espera 3s para o removedor conseguir remover a peça. Se o botão de STOP estiver pressionado, não reinicia o sistema de separação (Etapa 0). Senão reinicia (Etapa 99). *)
_e10(CLK := 28 = Etapas);
IF _e10.Q THEN Inc(InOut := LidCountAux); END_IF;
timer_S12(In := 28 = Etapas, PT := t#3s);
IF timer_S12.Q THEN Etapas := 92; END_IF;
(* notes on elements: Tempo de atividade do Remover de Peças Lid *)

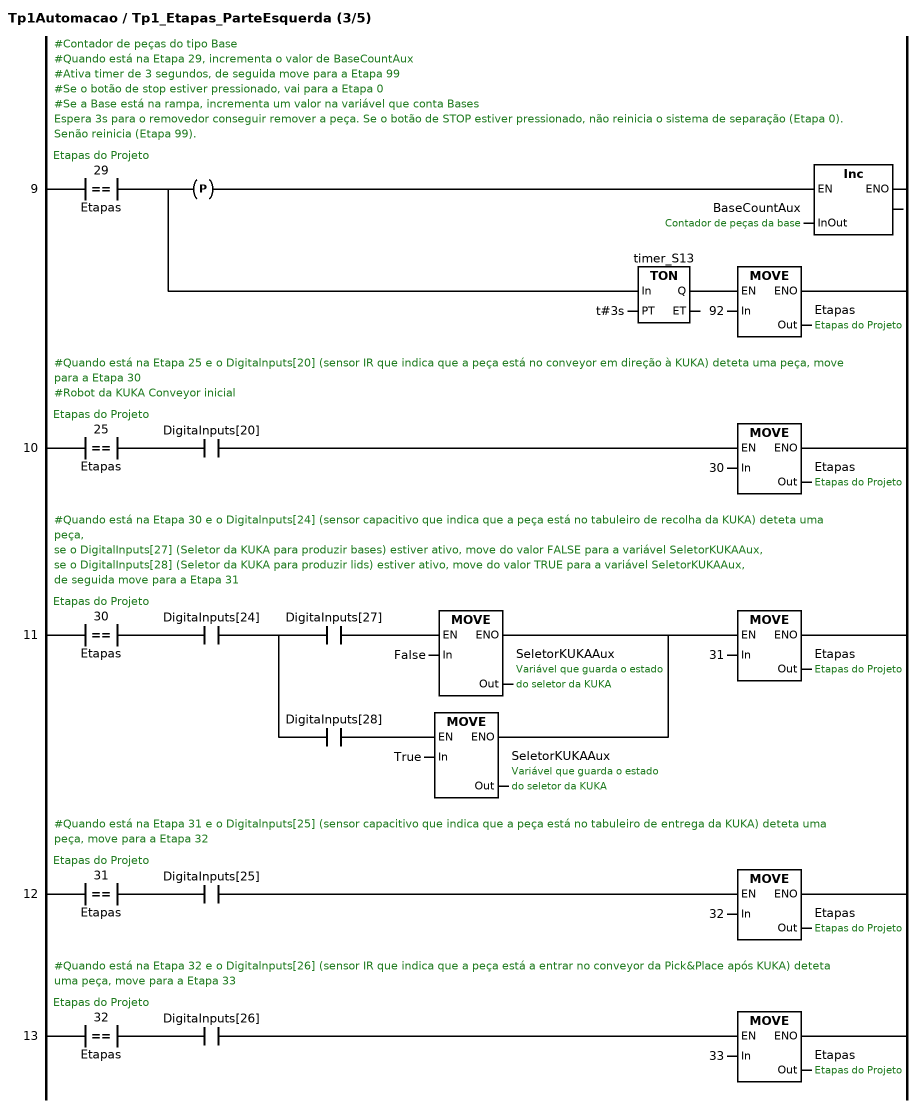
(* Rung 9: #Contador de peças do tipo Base / #Quando está na Etapa 29, incrementa o valor de BaseCountAux / #Ativa timer de 3 segundos, de seguida move para a Etapa 99 / #Se o botão de stop estiver pressionado, vai para a Etapa 0 / #Se a Base está na rampa, incrementa um valor na variável que conta Bases / Espera 3s para o removedor conseguir remover a peça. Se o botão de STOP estiver pressionado, não reinicia o sistema de separação (Etapa 0). Senão reinicia (Etapa 99). *)
_e11(CLK := 29 = Etapas);
IF _e11.Q THEN Inc(InOut := BaseCountAux); END_IF;
timer_S13(In := 29 = Etapas, PT := t#3s);
IF timer_S13.Q THEN Etapas := 92; END_IF;
(* notes on elements: Tempo de atividade do Remover de Peças Base *)
(* Rung 10: #Quando está na Etapa 25 e o Digitalnputs[20] (sensor IR que indica que a peça está no conveyor em direção à KUKA) deteta uma peça, move para a Etapa 30 / #Robot da KUKA Conveyor inicial *)
IF (25 = Etapas) AND DigitaInputs[20] THEN Etapas := 30; END_IF;
(* Rung 11: #Quando está na Etapa 30 e o Digitalnputs[24] (sensor capacitivo que indica que a peça está no tabuleiro de recolha da KUKA) deteta uma peça, / se o DigitalInputs[27] (Seletor da KUKA para produzir bases) estiver ativo, move do valor FALSE para a variável SeletorKUKAAux, / se o DigitalInputs[28] (Seletor da KUKA para produzir lids) estiver ativo, move do valor TRUE para a variável SeletorKUKAAux, / de seguida move para a Etapa 31 *)
IF (30 = Etapas) AND DigitaInputs[24] AND DigitaInputs[27] THEN SeletorKUKAAux := False; END_IF;
IF (30 = Etapas) AND DigitaInputs[24] AND DigitaInputs[28] THEN SeletorKUKAAux := True; END_IF;
IF (30 = Etapas) AND DigitaInputs[24] AND (DigitaInputs[27] OR DigitaInputs[28]) THEN
    Etapas := 31;
END_IF;
(* Rung 12: #Quando está na Etapa 31 e o Digitalnputs[25] (sensor capacitivo que indica que a peça está no tabuleiro de entrega da KUKA) deteta uma peça, move para a Etapa 32 *)
IF (31 = Etapas) AND DigitaInputs[25] THEN Etapas := 32; END_IF;
(* Rung 13: #Quando está na Etapa 32 e o Digitalnputs[26] (sensor IR que indica que a peça está a entrar no conveyor da Pick&Place após KUKA) deteta uma peça, move para a Etapa 33 *)
IF (32 = Etapas) AND DigitaInputs[26] THEN Etapas := 33; END_IF;

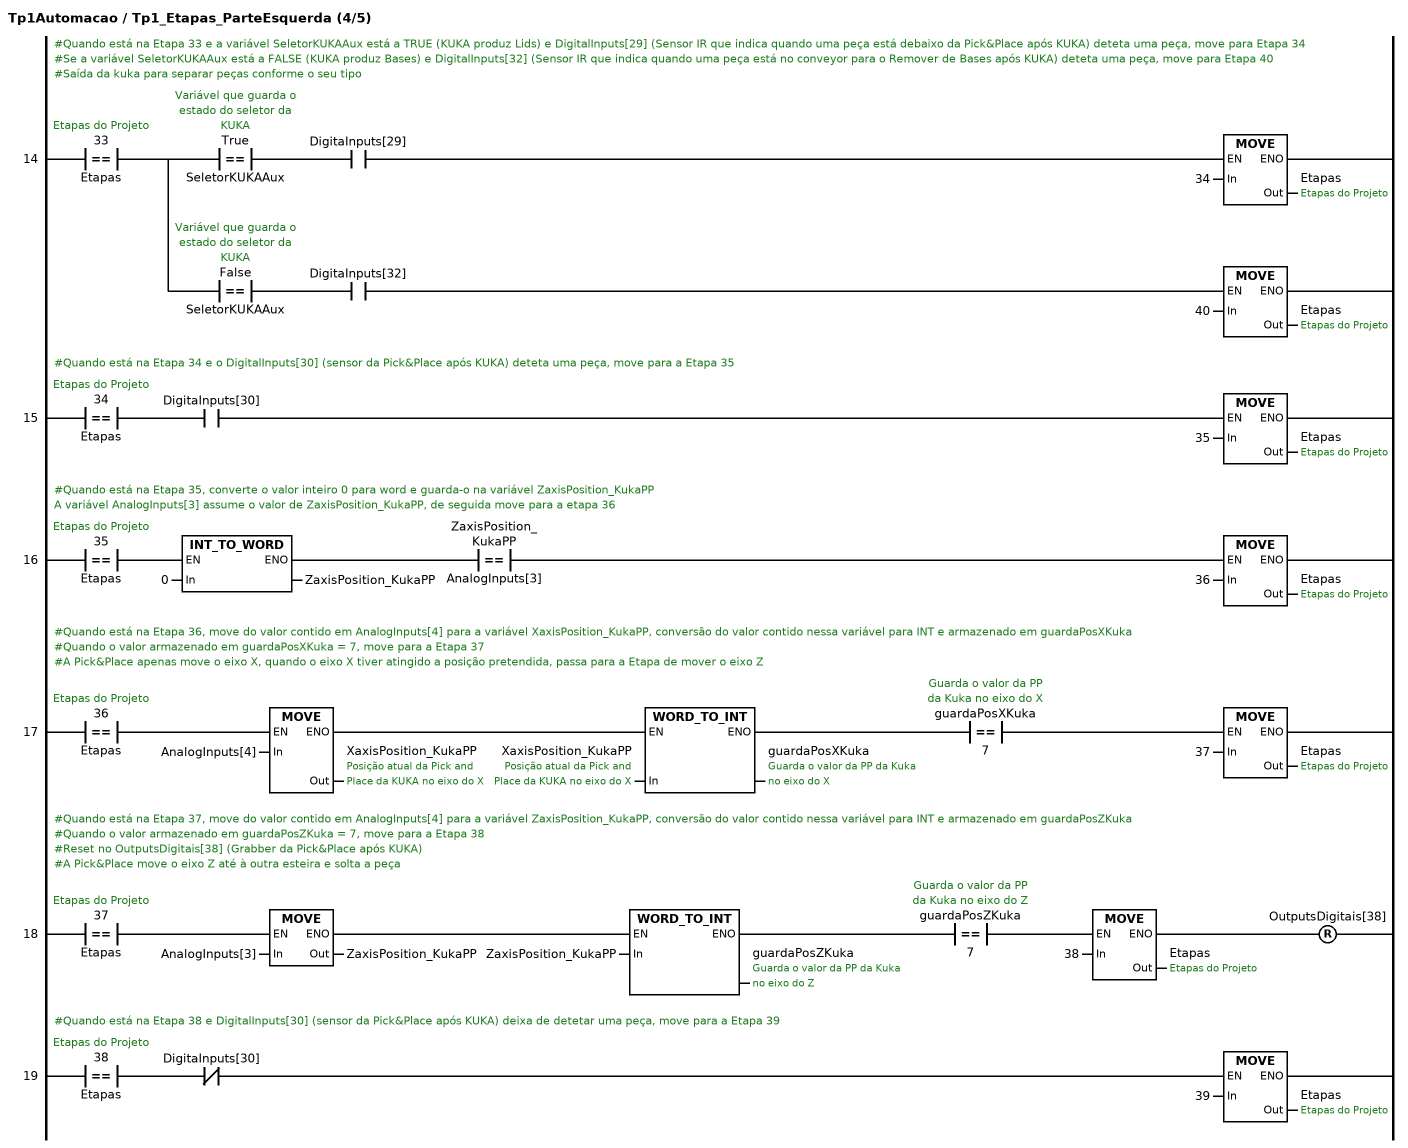
(* Rung 14: #Quando está na Etapa 33 e a variável SeletorKUKAAux está a TRUE (KUKA produz Lids) e DigitalInputs[29] (Sensor IR que indica quando uma peça está debaixo da Pick&Place após KUKA) deteta uma peça, move para Etapa 34 / #Se a variável SeletorKUKAAux está a FALSE (KUKA produz Bases) e DigitalInputs[32] (Sensor IR que indica quando uma peça está no conveyor para o Remover de Bases após KUKA) deteta uma peça, move para Etapa 40 / #Saída da kuka para separar peças conforme o seu tipo *)
_p12 := 33 = Etapas;
IF (33 = Etapas) AND (True = SeletorKUKAAux) AND DigitaInputs[29] THEN Etapas := 34; END_IF;
IF _p12 AND (False = SeletorKUKAAux) AND DigitaInputs[32] THEN Etapas := 40; END_IF;
(* Rung 15: #Quando está na Etapa 34 e o DigitalInputs[30] (sensor da Pick&Place após KUKA) deteta uma peça, move para a Etapa 35 *)
IF (34 = Etapas) AND DigitaInputs[30] THEN Etapas := 35; END_IF;
(* Rung 16: #Quando está na Etapa 35, converte o valor inteiro 0 para word e guarda-o na variável ZaxisPosition_KukaPP / A variável AnalogInputs[3] assume o valor de ZaxisPosition_KukaPP, de seguida move para a etapa 36 *)
IF 35 = Etapas THEN ZaxisPosition_KukaPP := INT_TO_WORD(In := 0); END_IF;
IF (35 = Etapas) AND (ZaxisPosition_KukaPP = AnalogInputs[3]) THEN Etapas := 36; END_IF;
(* Rung 17: #Quando está na Etapa 36, move do valor contido em AnalogInputs[4] para a variável XaxisPosition_KukaPP, conversão do valor contido nessa variável para INT e armazenado em guardaPosXKuka / #Quando o valor armazenado em guardaPosXKuka = 7, move para a Etapa 37 / #A Pick&Place apenas move o eixo X, quando o eixo X tiver atingido a posição pretendida, passa para a Etapa de mover o eixo Z *)
IF 36 = Etapas THEN
    XaxisPosition_KukaPP := AnalogInputs[4];
    guardaPosXKuka := WORD_TO_INT(In := XaxisPosition_KukaPP);
END_IF;
IF (36 = Etapas) AND (guardaPosXKuka = 7) THEN Etapas := 37; END_IF;
(* Rung 18: #Quando está na Etapa 37, move do valor contido em AnalogInputs[4] para a variável ZaxisPosition_KukaPP, conversão do valor contido nessa variável para INT e armazenado em guardaPosZKuka / #Quando o valor armazenado em guardaPosZKuka = 7, move para a Etapa 38 / #Reset no OutputsDigitais[38] (Grabber da Pick&Place após KUKA) / #A Pick&Place move o eixo Z até à outra esteira e solta a peça *)
IF 37 = Etapas THEN
    ZaxisPosition_KukaPP := AnalogInputs[3];
    guardaPosZKuka := WORD_TO_INT(In := ZaxisPosition_KukaPP);
END_IF;
_p13 := (37 = Etapas) AND (guardaPosZKuka = 7);
IF _p13 THEN
    Etapas := 38;
    OutputsDigitais[38] := FALSE;
END_IF;
(* Rung 19: #Quando está na Etapa 38 e DigitalInputs[30] (sensor da Pick&Place após KUKA) deixa de detetar uma peça, move para a Etapa 39 *)
IF (38 = Etapas) AND NOT DigitaInputs[30] THEN Etapas := 39; END_IF;

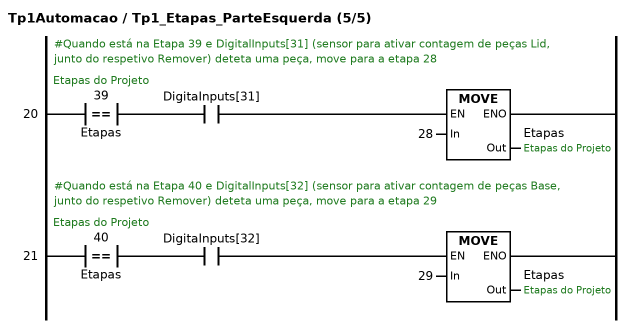
(* Rung 20: #Quando está na Etapa 39 e DigitalInputs[31] (sensor para ativar contagem de peças Lid, junto do respetivo Remover) deteta uma peça, move para a etapa 28 *)
IF (39 = Etapas) AND DigitaInputs[31] THEN Etapas := 28; END_IF;
(* Rung 21: #Quando está na Etapa 40 e DigitalInputs[32] (sensor para ativar contagem de peças Base, junto do respetivo Remover) deteta uma peça, move para a etapa 29 *)
IF (40 = Etapas) AND DigitaInputs[32] THEN Etapas := 29; END_IF;

(* Section Tp1_Outputs_ParteEsquerda: ladder, written here as Structured Text *)

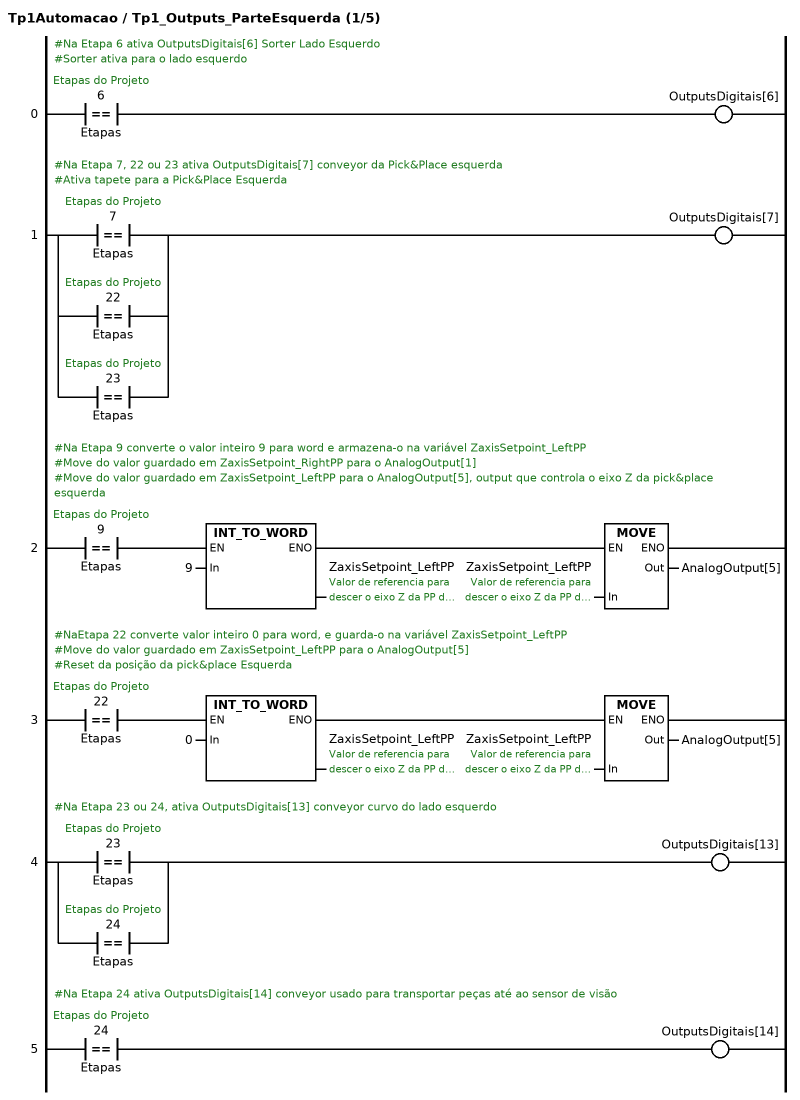
(* Rung 0: #Na Etapa 6 ativa OutputsDigitais[6] Sorter Lado Esquerdo / #Sorter ativa para o lado esquerdo *)
OutputsDigitais[6] := 6 = Etapas;
(* Rung 1: #Na Etapa 7, 22 ou 23 ativa OutputsDigitais[7] conveyor da Pick&Place esquerda / #Ativa tapete para a Pick&Place Esquerda *)
OutputsDigitais[7] := (7 = Etapas) OR (22 = Etapas) OR (23 = Etapas);
(* Rung 2: #Na Etapa 9 converte o valor inteiro 9 para word e armazena-o na variável ZaxisSetpoint_LeftPP / #Move do valor guardado em ZaxisSetpoint_RightPP para o AnalogOutput[1] / #Move do valor guardado em ZaxisSetpoint_LeftPP para o AnalogOutput[5], output que controla o eixo Z da pick&place esquerda *)
IF 9 = Etapas THEN
    ZaxisSetpoint_LeftPP := INT_TO_WORD(In := 9);
    AnalogOutput[5] := ZaxisSetpoint_LeftPP;
END_IF;
(* Rung 3: #NaEtapa 22 converte valor inteiro 0 para word, e guarda-o na variável ZaxisSetpoint_LeftPP / #Move do valor guardado em ZaxisSetpoint_LeftPP para o AnalogOutput[5] / #Reset da posição da pick&place Esquerda *)
IF 22 = Etapas THEN
    ZaxisSetpoint_LeftPP := INT_TO_WORD(In := 0);
    AnalogOutput[5] := ZaxisSetpoint_LeftPP;
END_IF;
(* Rung 4: #Na Etapa 23 ou 24, ativa OutputsDigitais[13] conveyor curvo do lado esquerdo *)
OutputsDigitais[13] := (23 = Etapas) OR (24 = Etapas);
(* Rung 5: #Na Etapa 24 ativa OutputsDigitais[14] conveyor usado para transportar peças até ao sensor de visão *)
OutputsDigitais[14] := 24 = Etapas;

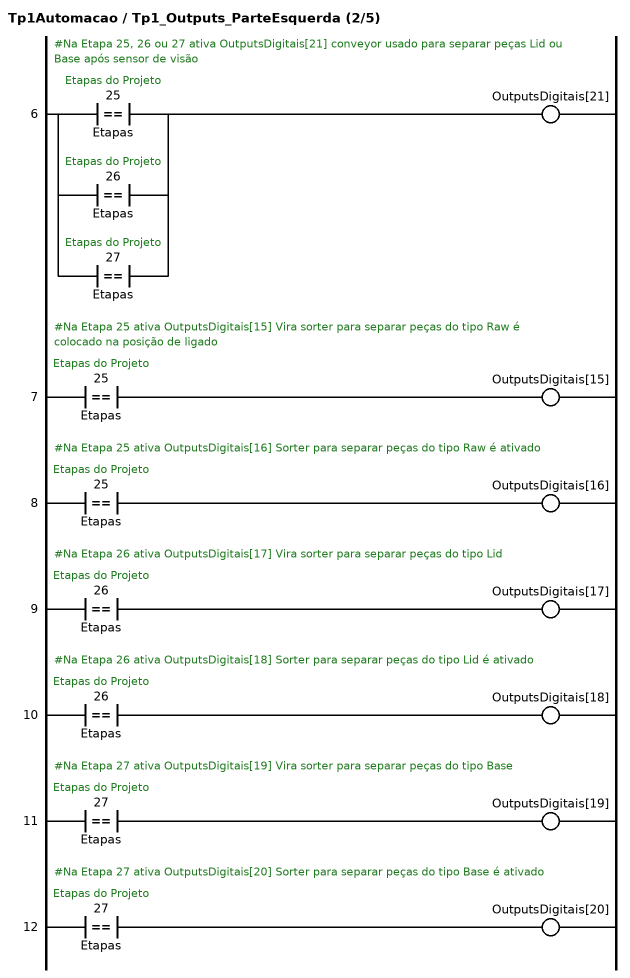
(* Rung 6: #Na Etapa 25, 26 ou 27 ativa OutputsDigitais[21] conveyor usado para separar peças Lid ou Base após sensor de visão *)
OutputsDigitais[21] := (25 = Etapas) OR (26 = Etapas) OR (27 = Etapas);
(* Rung 7: #Na Etapa 25 ativa OutputsDigitais[15] Vira sorter para separar peças do tipo Raw é colocado na posição de ligado *)
OutputsDigitais[15] := 25 = Etapas;
(* Rung 8: #Na Etapa 25 ativa OutputsDigitais[16] Sorter para separar peças do tipo Raw é ativado *)
OutputsDigitais[16] := 25 = Etapas;
(* Rung 9: #Na Etapa 26 ativa OutputsDigitais[17] Vira sorter para separar peças do tipo Lid *)
OutputsDigitais[17] := 26 = Etapas;
(* Rung 10: #Na Etapa 26 ativa OutputsDigitais[18] Sorter para separar peças do tipo Lid é ativado *)
OutputsDigitais[18] := 26 = Etapas;
(* Rung 11: #Na Etapa 27 ativa OutputsDigitais[19] Vira sorter para separar peças do tipo Base *)
OutputsDigitais[19] := 27 = Etapas;
(* Rung 12: #Na Etapa 27 ativa OutputsDigitais[20] Sorter para separar peças do tipo Base é ativado *)
OutputsDigitais[20] := 27 = Etapas;

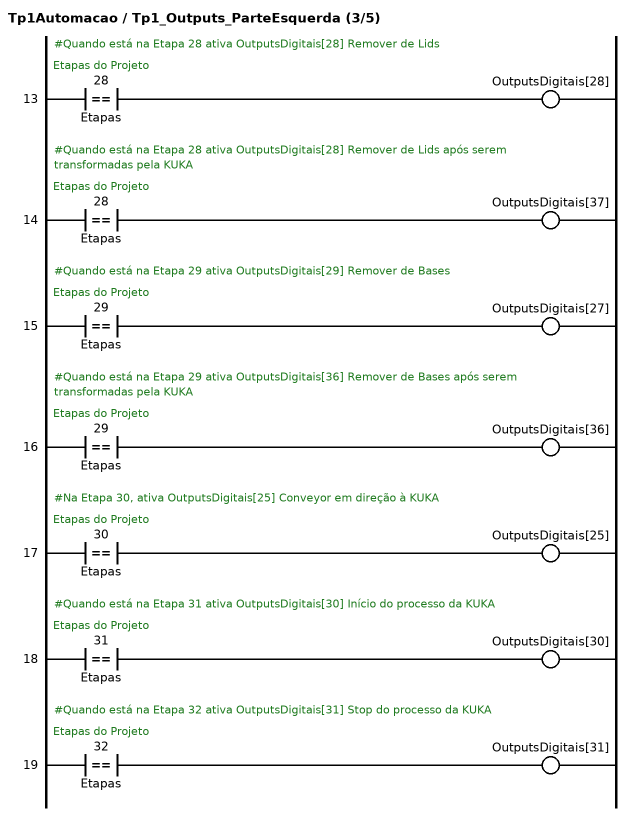
(* Rung 13: #Quando está na Etapa 28 ativa OutputsDigitais[28] Remover de Lids *)
OutputsDigitais[28] := 28 = Etapas;
(* Rung 14: #Quando está na Etapa 28 ativa OutputsDigitais[28] Remover de Lids após serem transformadas pela KUKA *)
OutputsDigitais[37] := 28 = Etapas;
(* Rung 15: #Quando está na Etapa 29 ativa OutputsDigitais[29] Remover de Bases *)
OutputsDigitais[27] := 29 = Etapas;
(* Rung 16: #Quando está na Etapa 29 ativa OutputsDigitais[36] Remover de Bases após serem transformadas pela KUKA *)
OutputsDigitais[36] := 29 = Etapas;
(* Rung 17: #Na Etapa 30, ativa OutputsDigitais[25] Conveyor em direção à KUKA *)
OutputsDigitais[25] := 30 = Etapas;
(* Rung 18: #Quando está na Etapa 31 ativa OutputsDigitais[30] Início do processo da KUKA *)
OutputsDigitais[30] := 31 = Etapas;
(* Rung 19: #Quando está na Etapa 32 ativa OutputsDigitais[31] Stop do processo da KUKA *)
OutputsDigitais[31] := 32 = Etapas;

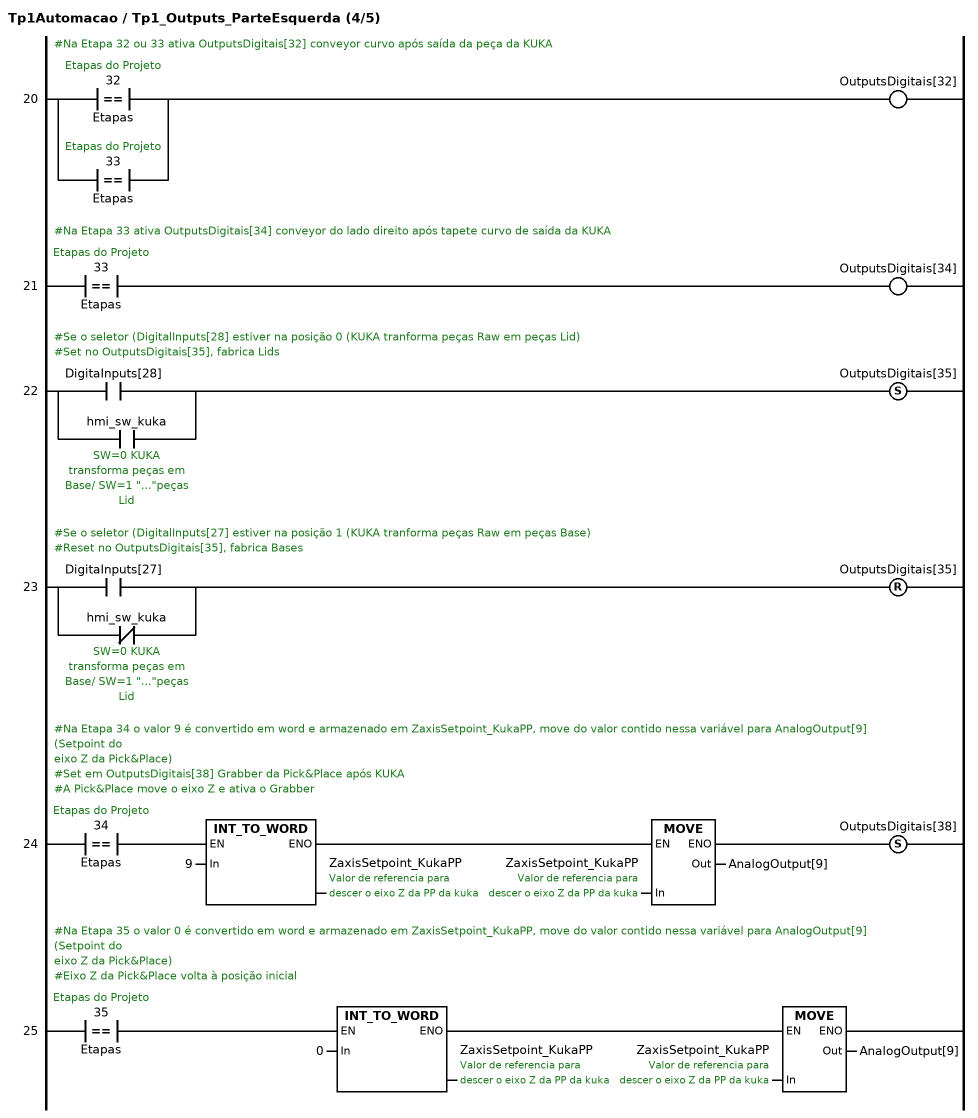
(* Rung 20: #Na Etapa 32 ou 33 ativa OutputsDigitais[32] conveyor curvo após saída da peça da KUKA *)
OutputsDigitais[32] := (32 = Etapas) OR (33 = Etapas);
(* Rung 21: #Na Etapa 33 ativa OutputsDigitais[34] conveyor do lado direito após tapete curvo de saída da KUKA *)
OutputsDigitais[34] := 33 = Etapas;
(* Rung 22: #Se o seletor (DigitalInputs[28] estiver na posição 0 (KUKA tranforma peças Raw em peças Lid) / #Set no OutputsDigitais[35], fabrica Lids *)
IF DigitaInputs[28] OR hmi_sw_kuka THEN OutputsDigitais[35] := TRUE; END_IF;
(* Rung 23: #Se o seletor (DigitalInputs[27] estiver na posição 1 (KUKA tranforma peças Raw em peças Base) / #Reset no OutputsDigitais[35], fabrica Bases *)
IF DigitaInputs[27] OR NOT hmi_sw_kuka THEN OutputsDigitais[35] := FALSE; END_IF;
(* Rung 24: #Na Etapa 34 o valor 9 é convertido em word e armazenado em ZaxisSetpoint_KukaPP, move do valor contido nessa variável para AnalogOutput[9] (Setpoint do / eixo Z da Pick&Place) / #Set em OutputsDigitais[38] Grabber da Pick&Place após KUKA / #A Pick&Place move o eixo Z e ativa o Grabber *)
IF 34 = Etapas THEN
    ZaxisSetpoint_KukaPP := INT_TO_WORD(In := 9);
    AnalogOutput[9] := ZaxisSetpoint_KukaPP;
    OutputsDigitais[38] := TRUE;
END_IF;
(* Rung 25: #Na Etapa 35 o valor 0 é convertido em word e armazenado em ZaxisSetpoint_KukaPP, move do valor contido nessa variável para AnalogOutput[9] (Setpoint do / eixo Z da Pick&Place) / #Eixo Z da Pick&Place volta à posição inicial *)
IF 35 = Etapas THEN
    ZaxisSetpoint_KukaPP := INT_TO_WORD(In := 0);
    AnalogOutput[9] := ZaxisSetpoint_KukaPP;
END_IF;

